KUKA KRL program: f1_Kuka_APT205T02S05.SRC

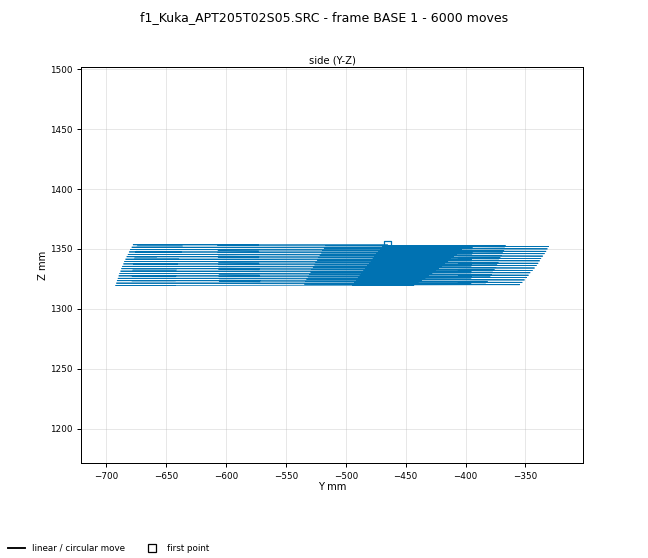
[picture p0: tool path of f1_Kuka_APT205T02S05.SRC in frame BASE 1, 6000 of 6001 moves have a stored position in this frame; points joined in program order, loops and branches not executed]
&ACCESS RVP
&REL 2
&PARAM TEMPLATE = C:\KRC\Roboter\Template\vorgabe
&PARAM EDITMASK = *
DEF f1_Kuka_APT205T02S05()


;FOLD INI;%{PE}%V3.2.0,%MKUKATPBASIS,%CINIT,%VCOMMON,%P
  ;FOLD BAS INI;%{E}%V3.2.0,%MKUKATPBASIS,%CINIT,%VINIT,%P
    GLOBAL INTERRUPT DECL 3 WHEN $STOPMESS==TRUE DO IR_STOPM ( )
    INTERRUPT ON 3
    BAS (#INITMOV,0 )
  ;ENDFOLD (BAS INI)
  ;FOLD USER INI;%{E}%V3.2.0,%MKUKATPUSER,%CINIT,%VINIT,%P
    ;Make your modifications here
  ;ENDFOLD (USER INI)
;ENDFOLD (INI)


;*** Make Null PTP Move
  PTP $pos_act

;*** Auto Load The Correct TOOL Data
  $tool=tool_data[2]

;*** Auto Load The Correct BASE Data
  $base=base_data[1]

  $ADVANCE = 5

;*** Restate Last Velocity
MMPM(30000.0)
SetRPM(8000)
LIN {X 0.183,Y -465.131,Z 1353.680,A 0.000,B 0.000,C 90.000,E1 158.284} C_DIS
LIN {X 0.167,Y -471.165,Z 1353.677,A 0.000,B 0.000,C 90.000,E1 157.794} C_DIS
LIN {X 0.121,Y -479.933,Z 1353.673,A 0.000,B 0.000,C 90.000,E1 157.050} C_DIS
LIN {X -0.013,Y -487.034,Z 1353.669,A 0.000,B 0.000,C 90.000,E1 156.433} C_DIS
LIN {X -0.242,Y -494.071,Z 1353.665,A 0.000,B 0.000,C 90.000,E1 155.793} C_DIS
LIN {X 0.180,Y -502.264,Z 1353.661,A 0.000,B 0.000,C 90.000,E1 154.921} C_DIS
LIN {X -0.273,Y -507.490,Z 1353.658,A 0.000,B 0.000,C 90.000,E1 154.409} C_DIS
LIN {X 0.116,Y -513.891,Z 1353.654,A 0.000,B 0.000,C 90.000,E1 153.640} C_DIS
LIN {X -0.118,Y -518.707,Z 1353.650,A 0.000,B 0.000,C 90.000,E1 153.076} C_DIS
LIN {X 0.081,Y -522.053,Z 1353.648,A 0.000,B 0.000,C 90.000,E1 152.615} C_DIS
LIN {X 0.144,Y -526.085,Z 1353.645,A 0.000,B 0.000,C 90.000,E1 152.025} C_DIS
LIN {X 0.240,Y -529.707,Z 1353.641,A 0.000,B 0.000,C 90.000,E1 151.435} C_DIS
LIN {X 0.217,Y -533.478,Z 1353.637,A 0.000,B 0.000,C 90.000,E1 150.717} C_DIS
LIN {X -0.096,Y -536.078,Z 1353.634,A 0.000,B 0.000,C 90.000,E1 150.177} C_DIS
LIN {X -0.207,Y -539.262,Z 1353.630,A 0.000,B 0.000,C 90.000,E1 149.331} C_DIS
LIN {X -0.021,Y -541.185,Z 1353.626,A 0.000,B 0.000,C 90.000,E1 148.742} C_DIS
LIN {X -0.285,Y -542.841,Z 1353.623,A 0.000,B 0.000,C 90.000,E1 148.201} C_DIS
LIN {X -0.054,Y -544.956,Z 1353.619,A 0.000,B 0.000,C 90.000,E1 147.327} C_DIS
LIN {X -0.260,Y -546.709,Z 1353.614,A 0.000,B 0.000,C 90.000,E1 146.501} C_DIS
LIN {X 0.272,Y -547.758,Z 1353.611,A 0.000,B 0.000,C 90.000,E1 145.881} C_DIS
LIN {X 0.097,Y -549.026,Z 1353.606,A 0.000,B 0.000,C 90.000,E1 145.055} C_DIS
LIN {X 0.251,Y -550.065,Z 1353.601,A 0.000,B 0.000,C 90.000,E1 144.196} C_DIS
LIN {X -0.292,Y -551.238,Z 1353.595,A 0.000,B 0.000,C 90.000,E1 143.130} C_DIS
LIN {X -0.048,Y -552.087,Z 1353.589,A 0.000,B 0.000,C 90.000,E1 141.984} C_DIS
LIN {X -0.168,Y -553.059,Z 1353.581,A 0.000,B 0.000,C 90.000,E1 140.598} C_DIS
LIN {X -0.278,Y -554.077,Z 1353.572,A 0.000,B 0.000,C 90.000,E1 138.933} C_DIS
LIN {X -0.078,Y -554.702,Z 1353.566,A 0.000,B 0.000,C 90.000,E1 137.796} C_DIS
LIN {X 0.097,Y -555.358,Z 1353.559,A 0.000,B 0.000,C 90.000,E1 136.662} C_DIS
LIN {X -0.235,Y -556.623,Z 1353.545,A 0.000,B 0.000,C 90.000,E1 134.190} C_DIS
LIN {X -0.134,Y -557.642,Z 1353.541,A 0.000,B 0.000,C 90.000,E1 133.299} C_DIS
LIN {X -0.120,Y -557.742,Z 1353.540,A 0.000,B 0.000,C 90.000,E1 133.257} C_DIS
LIN {X 0.206,Y -557.794,Z 1353.540,A 0.000,B 0.000,C 90.000,E1 133.218} C_DIS
LIN {X 0.099,Y -558.727,Z 1353.540,A 0.000,B 0.000,C 90.000,E1 133.137} C_DIS
LIN {X -0.091,Y -560.305,Z 1353.538,A 0.000,B 0.000,C 90.000,E1 132.894} C_DIS
LIN {X -0.316,Y -560.480,Z 1353.538,A 0.000,B 0.000,C 90.000,E1 132.852} C_DIS
LIN {X 0.022,Y -560.547,Z 1353.538,A 0.000,B 0.000,C 90.000,E1 132.813} C_DIS
LIN {X -0.018,Y -565.337,Z 1353.537,A 0.000,B 0.000,C 90.000,E1 132.609} C_DIS
LIN {X -0.209,Y -572.122,Z 1353.536,A 0.000,B 0.000,C 90.000,E1 132.447} C_DIS
LIN {X 0.152,Y -578.607,Z 1353.535,A 0.000,B 0.000,C 90.000,E1 132.204} C_DIS
LIN {X 0.195,Y -583.987,Z 1353.533,A 0.000,B 0.000,C 90.000,E1 131.919} C_DIS
LIN {X -0.113,Y -589.724,Z 1353.531,A 0.000,B 0.000,C 90.000,E1 131.595} C_DIS
LIN {X -0.223,Y -594.067,Z 1353.529,A 0.000,B 0.000,C 90.000,E1 131.310} C_DIS
LIN {X -0.123,Y -599.587,Z 1353.527,A 0.000,B 0.000,C 90.000,E1 130.862} C_DIS
LIN {X 0.104,Y -604.626,Z 1353.525,A 0.000,B 0.000,C 90.000,E1 130.415} C_DIS
LIN {X -0.052,Y -609.589,Z 1353.522,A 0.000,B 0.000,C 90.000,E1 129.967} C_DIS
LIN {X -0.137,Y -614.548,Z 1353.519,A 0.000,B 0.000,C 90.000,E1 129.483} C_DIS
LIN {X 0.107,Y -619.394,Z 1353.516,A 0.000,B 0.000,C 90.000,E1 128.955} C_DIS
LIN {X 0.250,Y -625.158,Z 1353.513,A 0.000,B 0.000,C 90.000,E1 128.302} C_DIS
LIN {X -0.237,Y -630.534,Z 1353.510,A 0.000,B 0.000,C 90.000,E1 127.729} C_DIS
LIN {X -0.014,Y -634.609,Z 1353.507,A 0.000,B 0.000,C 90.000,E1 127.202} C_DIS
LIN {X -0.289,Y -641.308,Z 1353.502,A 0.000,B 0.000,C 90.000,E1 126.377} C_DIS
LIN {X -0.064,Y -648.746,Z 1353.496,A 0.000,B 0.000,C 90.000,E1 125.358} C_DIS
LIN {X -0.070,Y -652.974,Z 1353.493,A 0.000,B 0.000,C 90.000,E1 124.739} C_DIS
LIN {X 0.045,Y -655.457,Z 1353.491,A 0.000,B 0.000,C 90.000,E1 124.358} C_DIS
LIN {X -0.290,Y -659.110,Z 1353.488,A 0.000,B 0.000,C 90.000,E1 123.785} C_DIS
LIN {X -0.210,Y -662.478,Z 1353.484,A 0.000,B 0.000,C 90.000,E1 123.166} C_DIS
LIN {X -0.165,Y -664.889,Z 1353.481,A 0.000,B 0.000,C 90.000,E1 122.673} C_DIS
LIN {X 0.027,Y -668.041,Z 1353.477,A 0.000,B 0.000,C 90.000,E1 121.926} C_DIS
LIN {X -0.101,Y -670.798,Z 1353.473,A 0.000,B 0.000,C 90.000,E1 121.209} C_DIS
LIN {X -0.265,Y -673.818,Z 1353.468,A 0.000,B 0.000,C 90.000,E1 120.256} C_DIS
LIN {X -0.330,Y -675.665,Z 1353.464,A 0.000,B 0.000,C 90.000,E1 119.539} C_DIS
LIN {X -0.374,Y -676.912,Z 1353.460,A 0.000,B 0.000,C 90.000,E1 118.821} C_DIS
LIN {X -0.404,Y -677.509,Z 1353.456,A 0.000,B 0.000,C 90.000,E1 118.103} C_DIS
LIN {X 0.173,Y -677.641,Z 1353.452,A 0.000,B 0.000,C 90.000,E1 117.334} C_DIS
LIN {X 0.338,Y -677.452,Z 1353.447,A 0.000,B 0.000,C 90.000,E1 116.360} C_DIS
LIN {X 0.010,Y -677.039,Z 1353.443,A 0.000,B 0.000,C 90.000,E1 115.668} C_DIS
LIN {X -0.034,Y -676.246,Z 1353.439,A 0.000,B 0.000,C 90.000,E1 114.951} C_DIS
LIN {X 0.055,Y -675.448,Z 1353.436,A 0.000,B 0.000,C 90.000,E1 114.463} C_DIS
LIN {X -0.195,Y -673.854,Z 1353.433,A 0.000,B 0.000,C 90.000,E1 114.003} C_DIS
LIN {X -0.289,Y -672.736,Z 1353.432,A 0.000,B 0.000,C 90.000,E1 113.770} C_DIS
LIN {X 0.053,Y -669.200,Z 1353.429,A 0.000,B 0.000,C 90.000,E1 113.259} C_DIS
LIN {X 0.132,Y -667.975,Z 1353.429,A 0.000,B 0.000,C 90.000,E1 113.131} C_DIS
LIN {X 0.067,Y -661.845,Z 1353.426,A 0.000,B 0.000,C 90.000,E1 112.717} C_DIS
LIN {X -0.202,Y -659.937,Z 1353.426,A 0.000,B 0.000,C 90.000,E1 112.642} C_DIS
LIN {X 0.198,Y -653.354,Z 1353.425,A 0.000,B 0.000,C 90.000,E1 112.386} C_DIS
LIN {X 0.212,Y -645.926,Z 1353.423,A 0.000,B 0.000,C 90.000,E1 112.206} C_DIS
LIN {X 0.189,Y -635.486,Z 1353.422,A 0.000,B 0.000,C 90.000,E1 111.972} C_DIS
LIN {X 0.137,Y -635.322,Z 1353.422,A 0.000,B 0.000,C 90.000,E1 111.972} C_DIS
LIN {X -0.263,Y -636.382,Z 1353.421,A 0.000,B 0.000,C 90.000,E1 111.844} C_DIS
LIN {X 0.284,Y -644.889,Z 1353.416,A 0.000,B 0.000,C 90.000,E1 110.791} C_DIS
LIN {X 0.217,Y -649.631,Z 1353.412,A 0.000,B 0.000,C 90.000,E1 110.174} C_DIS
LIN {X 0.007,Y -654.094,Z 1353.408,A 0.000,B 0.000,C 90.000,E1 109.450} C_DIS
LIN {X -0.159,Y -657.809,Z 1353.404,A 0.000,B 0.000,C 90.000,E1 108.725} C_DIS
LIN {X -0.293,Y -661.030,Z 1353.400,A 0.000,B 0.000,C 90.000,E1 108.000} C_DIS
LIN {X 0.141,Y -664.980,Z 1353.395,A 0.000,B 0.000,C 90.000,E1 106.985} C_DIS
LIN {X 0.157,Y -666.754,Z 1353.392,A 0.000,B 0.000,C 90.000,E1 106.496} C_DIS
LIN {X -0.083,Y -669.107,Z 1353.388,A 0.000,B 0.000,C 90.000,E1 105.788} C_DIS
LIN {X -0.158,Y -669.814,Z 1353.386,A 0.000,B 0.000,C 90.000,E1 105.552} C_DIS
LIN {X -0.190,Y -671.501,Z 1353.382,A 0.000,B 0.000,C 90.000,E1 104.828} C_DIS
LIN {X 0.331,Y -672.524,Z 1353.380,A 0.000,B 0.000,C 90.000,E1 104.300} C_DIS
LIN {X 0.209,Y -673.257,Z 1353.377,A 0.000,B 0.000,C 90.000,E1 103.828} C_DIS
LIN {X 0.035,Y -673.939,Z 1353.373,A 0.000,B 0.000,C 90.000,E1 103.119} C_DIS
LIN {X -0.081,Y -674.212,Z 1353.370,A 0.000,B 0.000,C 90.000,E1 102.647} C_DIS
LIN {X 0.267,Y -674.154,Z 1353.366,A 0.000,B 0.000,C 90.000,E1 101.895} C_DIS
LIN {X 0.096,Y -673.684,Z 1353.362,A 0.000,B 0.000,C 90.000,E1 101.186} C_DIS
LIN {X -0.026,Y -673.153,Z 1353.360,A 0.000,B 0.000,C 90.000,E1 100.715} C_DIS
LIN {X -0.211,Y -672.846,Z 1353.358,A 0.000,B 0.000,C 90.000,E1 100.489} C_DIS
LIN {X 0.321,Y -671.939,Z 1353.356,A 0.000,B 0.000,C 90.000,E1 99.962} C_DIS
LIN {X 0.069,Y -670.767,Z 1353.353,A 0.000,B 0.000,C 90.000,E1 99.500} C_DIS
LIN {X -0.003,Y -670.111,Z 1353.352,A 0.000,B 0.000,C 90.000,E1 99.265} C_DIS
LIN {X -0.261,Y -668.546,Z 1353.349,A 0.000,B 0.000,C 90.000,E1 98.803} C_DIS
LIN {X 0.230,Y -666.752,Z 1353.346,A 0.000,B 0.000,C 90.000,E1 98.276} C_DIS
LIN {X -0.236,Y -663.690,Z 1353.342,A 0.000,B 0.000,C 90.000,E1 97.587} C_DIS
LIN {X 0.114,Y -660.735,Z 1353.339,A 0.000,B 0.000,C 90.000,E1 96.947} C_DIS
LIN {X 0.151,Y -656.334,Z 1353.334,A 0.000,B 0.000,C 90.000,E1 96.087} C_DIS
LIN {X -0.295,Y -652.814,Z 1353.331,A 0.000,B 0.000,C 90.000,E1 95.511} C_DIS
LIN {X -0.282,Y -647.351,Z 1353.326,A 0.000,B 0.000,C 90.000,E1 94.645} C_DIS
LIN {X -0.274,Y -642.136,Z 1353.322,A 0.000,B 0.000,C 90.000,E1 93.898} C_DIS
LIN {X -0.111,Y -638.342,Z 1353.319,A 0.000,B 0.000,C 90.000,E1 93.383} C_DIS
LIN {X -0.031,Y -632.660,Z 1353.315,A 0.000,B 0.000,C 90.000,E1 92.751} C_DIS
LIN {X -0.038,Y -622.818,Z 1353.310,A 0.000,B 0.000,C 90.000,E1 91.776} C_DIS
LIN {X 0.147,Y -616.480,Z 1353.307,A 0.000,B 0.000,C 90.000,E1 91.146} C_DIS
LIN {X -0.106,Y -609.537,Z 1353.303,A 0.000,B 0.000,C 90.000,E1 90.573} C_DIS
LIN {X 0.254,Y -603.296,Z 1353.301,A 0.000,B 0.000,C 90.000,E1 90.115} C_DIS
LIN {X 0.236,Y -598.176,Z 1353.299,A 0.000,B 0.000,C 90.000,E1 89.828} C_DIS
LIN {X 0.187,Y -594.693,Z 1353.298,A 0.000,B 0.000,C 90.000,E1 89.656} C_DIS
LIN {X 0.205,Y -581.240,Z 1353.295,A 0.000,B 0.000,C 90.000,E1 89.083} C_DIS
LIN {X 0.020,Y -578.376,Z 1353.294,A 0.000,B 0.000,C 90.000,E1 88.969} C_DIS
LIN {X 0.191,Y -575.836,Z 1353.293,A 0.000,B 0.000,C 90.000,E1 88.797} C_DIS
LIN {X -0.266,Y -574.481,Z 1353.293,A 0.000,B 0.000,C 90.000,E1 88.740} C_DIS
LIN {X -0.147,Y -573.606,Z 1353.292,A 0.000,B 0.000,C 90.000,E1 88.625} C_DIS
LIN {X -0.152,Y -573.255,Z 1353.292,A 0.000,B 0.000,C 90.000,E1 88.568} C_DIS
LIN {X -0.137,Y -573.024,Z 1353.291,A 0.000,B 0.000,C 90.000,E1 88.453} C_DIS
LIN {X -0.080,Y -572.878,Z 1353.290,A 0.000,B 0.000,C 90.000,E1 88.165} C_DIS
LIN {X -0.016,Y -573.318,Z 1353.286,A 0.000,B 0.000,C 90.000,E1 87.478} C_DIS
LIN {X -0.115,Y -575.111,Z 1353.275,A 0.000,B 0.000,C 90.000,E1 85.584} C_DIS
LIN {X 0.078,Y -577.539,Z 1353.263,A 0.000,B 0.000,C 90.000,E1 83.394} C_DIS
LIN {X -0.026,Y -579.410,Z 1353.254,A 0.000,B 0.000,C 90.000,E1 81.781} C_DIS
LIN {X -0.153,Y -581.083,Z 1353.247,A 0.000,B 0.000,C 90.000,E1 80.443} C_DIS
LIN {X 0.090,Y -582.298,Z 1353.241,A 0.000,B 0.000,C 90.000,E1 79.342} C_DIS
LIN {X 0.124,Y -583.632,Z 1353.233,A 0.000,B 0.000,C 90.000,E1 77.993} C_DIS
LIN {X 0.184,Y -584.854,Z 1353.226,A 0.000,B 0.000,C 90.000,E1 76.645} C_DIS
LIN {X -0.165,Y -585.974,Z 1353.219,A 0.000,B 0.000,C 90.000,E1 75.338} C_DIS
LIN {X -0.169,Y -586.736,Z 1353.213,A 0.000,B 0.000,C 90.000,E1 74.267} C_DIS
LIN {X 0.165,Y -587.915,Z 1353.202,A 0.000,B 0.000,C 90.000,E1 72.362} C_DIS
LIN {X 0.031,Y -588.687,Z 1353.195,A 0.000,B 0.000,C 90.000,E1 71.040} C_DIS
LIN {X -0.023,Y -589.671,Z 1353.186,A 0.000,B 0.000,C 90.000,E1 69.444} C_DIS
LIN {X -0.059,Y -591.222,Z 1353.172,A 0.000,B 0.000,C 90.000,E1 67.050} C_DIS
LIN {X 0.057,Y -592.676,Z 1353.162,A 0.000,B 0.000,C 90.000,E1 65.177} C_DIS
LIN {X -0.334,Y -593.414,Z 1353.156,A 0.000,B 0.000,C 90.000,E1 64.152} C_DIS
LIN {X -0.004,Y -594.376,Z 1353.149,A 0.000,B 0.000,C 90.000,E1 62.794} C_DIS
LIN {X 0.081,Y -596.127,Z 1353.137,A 0.000,B 0.000,C 90.000,E1 60.667} C_DIS
LIN {X 0.272,Y -598.255,Z 1353.125,A 0.000,B 0.000,C 90.000,E1 58.535} C_DIS
LIN {X 0.185,Y -599.776,Z 1353.117,A 0.000,B 0.000,C 90.000,E1 56.962} C_DIS
LIN {X -0.018,Y -600.796,Z 1353.111,A 0.000,B 0.000,C 90.000,E1 55.928} C_DIS
LIN {X 0.038,Y -602.054,Z 1353.103,A 0.000,B 0.000,C 90.000,E1 54.609} C_DIS
LIN {X 0.136,Y -603.753,Z 1353.093,A 0.000,B 0.000,C 90.000,E1 52.763} C_DIS
LIN {X -0.152,Y -604.595,Z 1353.087,A 0.000,B 0.000,C 90.000,E1 51.743} C_DIS
LIN {X 0.092,Y -605.607,Z 1353.079,A 0.000,B 0.000,C 90.000,E1 50.150} C_DIS
LIN {X 0.207,Y -606.155,Z 1353.073,A 0.000,B 0.000,C 90.000,E1 49.094} C_DIS
LIN {X -0.124,Y -606.527,Z 1353.067,A 0.000,B 0.000,C 90.000,E1 48.081} C_DIS
LIN {X -0.192,Y -606.838,Z 1353.060,A 0.000,B 0.000,C 90.000,E1 46.782} C_DIS
LIN {X -0.042,Y -606.960,Z 1353.051,A 0.000,B 0.000,C 90.000,E1 45.202} C_DIS
LIN {X -0.368,Y -606.826,Z 1353.045,A 0.000,B 0.000,C 90.000,E1 44.190} C_DIS
LIN {X 0.171,Y -606.456,Z 1353.040,A 0.000,B 0.000,C 90.000,E1 43.095} C_DIS
LIN {X -0.087,Y -605.775,Z 1353.031,A 0.000,B 0.000,C 90.000,E1 41.553} C_DIS
LIN {X 0.038,Y -605.198,Z 1353.025,A 0.000,B 0.000,C 90.000,E1 40.496} C_DIS
LIN {X 0.206,Y -604.342,Z 1353.016,A 0.000,B 0.000,C 90.000,E1 38.910} C_DIS
LIN {X 0.181,Y -603.425,Z 1353.009,A 0.000,B 0.000,C 90.000,E1 37.604} C_DIS
LIN {X -0.115,Y -602.354,Z 1353.003,A 0.000,B 0.000,C 90.000,E1 36.583} C_DIS
LIN {X 0.391,Y -601.707,Z 1353.000,A 0.000,B 0.000,C 90.000,E1 36.011} C_DIS
LIN {X 0.299,Y -600.464,Z 1352.996,A 0.000,B 0.000,C 90.000,E1 35.231} C_DIS
LIN {X 0.093,Y -598.433,Z 1352.990,A 0.000,B 0.000,C 90.000,E1 34.199} C_DIS
LIN {X -0.037,Y -596.783,Z 1352.986,A 0.000,B 0.000,C 90.000,E1 33.420} C_DIS
LIN {X 0.205,Y -594.246,Z 1352.980,A 0.000,B 0.000,C 90.000,E1 32.339} C_DIS
LIN {X 0.210,Y -592.058,Z 1352.975,A 0.000,B 0.000,C 90.000,E1 31.544} C_DIS
LIN {X -0.122,Y -588.527,Z 1352.969,A 0.000,B 0.000,C 90.000,E1 30.512} C_DIS
LIN {X 0.158,Y -586.676,Z 1352.967,A 0.000,B 0.000,C 90.000,E1 29.951} C_DIS
LIN {X 0.090,Y -583.481,Z 1352.962,A 0.000,B 0.000,C 90.000,E1 29.155} C_DIS
LIN {X -0.151,Y -578.574,Z 1352.956,A 0.000,B 0.000,C 90.000,E1 28.103} C_DIS
LIN {X 0.037,Y -573.018,Z 1352.950,A 0.000,B 0.000,C 90.000,E1 27.001} C_DIS
LIN {X 0.145,Y -569.164,Z 1352.946,A 0.000,B 0.000,C 90.000,E1 26.309} C_DIS
LIN {X 0.047,Y -565.823,Z 1352.943,A 0.000,B 0.000,C 90.000,E1 25.771} C_DIS
LIN {X 0.091,Y -561.388,Z 1352.939,A 0.000,B 0.000,C 90.000,E1 25.079} C_DIS
LIN {X 0.300,Y -558.527,Z 1352.937,A 0.000,B 0.000,C 90.000,E1 24.643} C_DIS
LIN {X 0.279,Y -553.466,Z 1352.933,A 0.000,B 0.000,C 90.000,E1 23.951} C_DIS
LIN {X 0.211,Y -548.153,Z 1352.929,A 0.000,B 0.000,C 90.000,E1 23.259} C_DIS
LIN {X -0.105,Y -542.387,Z 1352.926,A 0.000,B 0.000,C 90.000,E1 22.589} C_DIS
LIN {X -0.051,Y -533.794,Z 1352.920,A 0.000,B 0.000,C 90.000,E1 21.589} C_DIS
LIN {X -0.220,Y -523.413,Z 1352.914,A 0.000,B 0.000,C 90.000,E1 20.482} C_DIS
LIN {X 0.087,Y -511.582,Z 1352.907,A 0.000,B 0.000,C 90.000,E1 19.214} C_DIS
LIN {X -0.134,Y -503.938,Z 1352.902,A 0.000,B 0.000,C 90.000,E1 18.417} C_DIS
LIN {X 0.088,Y -493.051,Z 1352.896,A 0.000,B 0.000,C 90.000,E1 17.275} C_DIS
LIN {X 0.155,Y -482.910,Z 1352.891,A 0.000,B 0.000,C 90.000,E1 16.315} C_DIS
LIN {X -0.050,Y -466.107,Z 1352.882,A 0.000,B 0.000,C 90.000,E1 14.717} C_DIS
LIN {X -0.017,Y -454.626,Z 1352.875,A 0.000,B 0.000,C 90.000,E1 13.592} C_DIS
LIN {X 0.099,Y -434.707,Z 1352.864,A 0.000,B 0.000,C 90.000,E1 11.535} C_DIS
LIN {X 0.038,Y -419.253,Z 1352.855,A 0.000,B 0.000,C 90.000,E1 9.849} C_DIS
LIN {X 0.108,Y -408.120,Z 1352.848,A 0.000,B 0.000,C 90.000,E1 8.568} C_DIS
LIN {X 0.156,Y -399.605,Z 1352.842,A 0.000,B 0.000,C 90.000,E1 7.587} C_DIS
LIN {X -0.151,Y -396.843,Z 1352.840,A 0.000,B 0.000,C 90.000,E1 7.296} C_DIS
LIN {X -0.035,Y -394.063,Z 1352.838,A 0.000,B 0.000,C 90.000,E1 6.834} C_DIS
LIN {X -0.072,Y -394.049,Z 1352.838,A 0.000,B 0.000,C 90.000,E1 6.834} C_DIS
LIN {X 0.040,Y -394.965,Z 1352.837,A 0.000,B 0.000,C 90.000,E1 6.663} C_DIS
LIN {X -0.100,Y -398.981,Z 1352.835,A 0.000,B 0.000,C 90.000,E1 6.315} C_DIS
LIN {X -0.090,Y -412.650,Z 1352.830,A 0.000,B 0.000,C 90.000,E1 5.334} C_DIS
LIN {X -0.158,Y -415.923,Z 1352.828,A 0.000,B 0.000,C 90.000,E1 5.106} C_DIS
LIN {X -0.168,Y -423.370,Z 1352.825,A 0.000,B 0.000,C 90.000,E1 4.473} C_DIS
LIN {X -0.125,Y -429.177,Z 1352.822,A 0.000,B 0.000,C 90.000,E1 3.898} C_DIS
LIN {X -0.204,Y -436.191,Z 1352.817,A 0.000,B 0.000,C 90.000,E1 3.151} C_DIS
LIN {X -0.062,Y -442.966,Z 1352.813,A 0.000,B 0.000,C 90.000,E1 2.350} C_DIS
LIN {X -0.089,Y -448.332,Z 1352.810,A 0.000,B 0.000,C 90.000,E1 1.718} C_DIS
LIN {X -0.125,Y -454.577,Z 1352.805,A 0.000,B 0.000,C 90.000,E1 0.917} C_DIS
LIN {X -0.227,Y -459.308,Z 1352.802,A 0.000,B 0.000,C 90.000,E1 0.286} C_DIS
LIN {X 0.027,Y -465.795,Z 1352.796,A 0.000,B 0.000,C 90.000,E1 359.312} C_DIS
LIN {X 0.129,Y -470.852,Z 1352.792,A 0.000,B 0.000,C 90.000,E1 358.511} C_DIS
LIN {X -0.047,Y -476.329,Z 1352.787,A 0.000,B 0.000,C 90.000,E1 357.593} C_DIS
LIN {X 0.014,Y -479.818,Z 1352.783,A 0.000,B 0.000,C 90.000,E1 356.963} C_DIS
LIN {X -0.209,Y -483.851,Z 1352.779,A 0.000,B 0.000,C 90.000,E1 356.216} C_DIS
LIN {X -0.062,Y -486.825,Z 1352.776,A 0.000,B 0.000,C 90.000,E1 355.584} C_DIS
LIN {X -0.221,Y -490.207,Z 1352.771,A 0.000,B 0.000,C 90.000,E1 354.837} C_DIS
LIN {X -0.024,Y -492.765,Z 1352.768,A 0.000,B 0.000,C 90.000,E1 354.204} C_DIS
LIN {X 0.088,Y -496.185,Z 1352.763,A 0.000,B 0.000,C 90.000,E1 353.280} C_DIS
LIN {X 0.239,Y -499.354,Z 1352.758,A 0.000,B 0.000,C 90.000,E1 352.356} C_DIS
LIN {X 0.156,Y -500.373,Z 1352.756,A 0.000,B 0.000,C 90.000,E1 352.064} C_DIS
LIN {X -0.143,Y -502.907,Z 1352.751,A 0.000,B 0.000,C 90.000,E1 351.197} C_DIS
LIN {X 0.078,Y -505.288,Z 1352.746,A 0.000,B 0.000,C 90.000,E1 350.274} C_DIS
LIN {X -0.139,Y -508.072,Z 1352.739,A 0.000,B 0.000,C 90.000,E1 349.106} C_DIS
LIN {X 0.224,Y -509.966,Z 1352.734,A 0.000,B 0.000,C 90.000,E1 348.173} C_DIS
LIN {X 0.108,Y -511.644,Z 1352.729,A 0.000,B 0.000,C 90.000,E1 347.297} C_DIS
LIN {X 0.124,Y -513.042,Z 1352.725,A 0.000,B 0.000,C 90.000,E1 346.408} C_DIS
LIN {X 0.133,Y -514.692,Z 1352.718,A 0.000,B 0.000,C 90.000,E1 345.227} C_DIS
LIN {X 0.188,Y -515.655,Z 1352.713,A 0.000,B 0.000,C 90.000,E1 344.338} C_DIS
LIN {X -0.244,Y -516.324,Z 1352.708,A 0.000,B 0.000,C 90.000,E1 343.504} C_DIS
LIN {X -0.024,Y -516.755,Z 1352.703,A 0.000,B 0.000,C 90.000,E1 342.598} C_DIS
LIN {X 0.042,Y -516.921,Z 1352.698,A 0.000,B 0.000,C 90.000,E1 341.710} C_DIS
LIN {X -0.222,Y -516.779,Z 1352.694,A 0.000,B 0.000,C 90.000,E1 340.859} C_DIS
LIN {X -0.090,Y -516.613,Z 1352.692,A 0.000,B 0.000,C 90.000,E1 340.550} C_DIS
LIN {X 0.043,Y -516.273,Z 1352.690,A 0.000,B 0.000,C 90.000,E1 340.242} C_DIS
LIN {X 0.176,Y -515.763,Z 1352.689,A 0.000,B 0.000,C 90.000,E1 339.934} C_DIS
LIN {X 0.130,Y -514.975,Z 1352.687,A 0.000,B 0.000,C 90.000,E1 339.645} C_DIS
LIN {X -0.223,Y -513.741,Z 1352.685,A 0.000,B 0.000,C 90.000,E1 339.390} C_DIS
LIN {X 0.081,Y -512.783,Z 1352.685,A 0.000,B 0.000,C 90.000,E1 339.209} C_DIS
LIN {X -0.095,Y -510.810,Z 1352.684,A 0.000,B 0.000,C 90.000,E1 339.082} C_DIS
LIN {X -0.228,Y -481.772,Z 1352.677,A 0.000,B 0.000,C 90.000,E1 337.794} C_DIS
LIN {X 0.049,Y -453.227,Z 1352.668,A 0.000,B 0.000,C 90.000,E1 336.305} C_DIS
LIN {X 0.187,Y -428.324,Z 1352.660,A 0.000,B 0.000,C 90.000,E1 334.845} C_DIS
LIN {X -0.103,Y -405.367,Z 1352.652,A 0.000,B 0.000,C 90.000,E1 333.384} C_DIS
LIN {X 0.001,Y -384.338,Z 1352.643,A 0.000,B 0.000,C 90.000,E1 331.820} C_DIS
LIN {X 0.190,Y -366.662,Z 1352.635,A 0.000,B 0.000,C 90.000,E1 330.333} C_DIS
LIN {X 0.162,Y -366.645,Z 1352.635,A 0.000,B 0.000,C 90.000,E1 330.333} C_DIS
LIN {X -0.069,Y -371.456,Z 1352.603,A 0.000,B 0.000,C 90.000,E1 324.562} C_DIS
LIN {X -0.081,Y -371.815,Z 1352.601,A 0.000,B 0.000,C 90.000,E1 324.196} C_DIS
LIN {X -0.013,Y -377.467,Z 1352.567,A 0.000,B 0.000,C 90.000,E1 317.957} C_DIS
LIN {X -0.027,Y -377.945,Z 1352.564,A 0.000,B 0.000,C 90.000,E1 317.595} C_DIS
LIN {X 0.001,Y -378.528,Z 1352.560,A 0.000,B 0.000,C 90.000,E1 316.863} C_DIS
LIN {X 0.023,Y -384.552,Z 1352.528,A 0.000,B 0.000,C 90.000,E1 311.067} C_DIS
LIN {X 0.068,Y -384.947,Z 1352.526,A 0.000,B 0.000,C 90.000,E1 310.701} C_DIS
LIN {X 0.016,Y -390.724,Z 1352.494,A 0.000,B 0.000,C 90.000,E1 304.978} C_DIS
LIN {X 0.083,Y -391.221,Z 1352.492,A 0.000,B 0.000,C 90.000,E1 304.612} C_DIS
LIN {X -0.110,Y -396.934,Z 1352.459,A 0.000,B 0.000,C 90.000,E1 298.615} C_DIS
LIN {X 0.190,Y -401.301,Z 1352.428,A 0.000,B 0.000,C 90.000,E1 292.950} C_DIS
LIN {X -0.100,Y -401.646,Z 1352.426,A 0.000,B 0.000,C 90.000,E1 292.642} C_DIS
LIN {X 0.036,Y -404.726,Z 1352.395,A 0.000,B 0.000,C 90.000,E1 287.040} C_DIS
LIN {X 0.039,Y -406.144,Z 1352.364,A 0.000,B 0.000,C 90.000,E1 281.478} C_DIS
LIN {X 0.137,Y -405.687,Z 1352.333,A 0.000,B 0.000,C 90.000,E1 275.910} C_DIS
LIN {X -0.195,Y -403.571,Z 1352.306,A 0.000,B 0.000,C 90.000,E1 271.088} C_DIS
LIN {X 0.144,Y -403.221,Z 1352.302,A 0.000,B 0.000,C 90.000,E1 270.344} C_DIS
LIN {X -0.022,Y -399.083,Z 1352.273,A 0.000,B 0.000,C 90.000,E1 265.122} C_DIS
LIN {X -0.080,Y -398.829,Z 1352.271,A 0.000,B 0.000,C 90.000,E1 264.780} C_DIS
LIN {X 0.206,Y -393.321,Z 1352.244,A 0.000,B 0.000,C 90.000,E1 259.803} C_DIS
LIN {X 0.127,Y -392.730,Z 1352.240,A 0.000,B 0.000,C 90.000,E1 259.106} C_DIS
LIN {X -0.180,Y -386.288,Z 1352.214,A 0.000,B 0.000,C 90.000,E1 254.519} C_DIS
LIN {X -0.109,Y -385.187,Z 1352.208,A 0.000,B 0.000,C 90.000,E1 253.433} C_DIS
LIN {X -0.142,Y -382.701,Z 1352.200,A 0.000,B 0.000,C 90.000,E1 252.000} C_DIS
LIN {X 0.113,Y -376.547,Z 1352.176,A 0.000,B 0.000,C 90.000,E1 247.614} C_DIS
LIN {X -0.109,Y -376.137,Z 1352.174,A 0.000,B 0.000,C 90.000,E1 247.283} C_DIS
LIN {X 0.063,Y -368.301,Z 1352.147,A 0.000,B 0.000,C 90.000,E1 242.487} C_DIS
LIN {X 0.100,Y -366.444,Z 1352.139,A 0.000,B 0.000,C 90.000,E1 241.001} C_DIS
LIN {X -0.135,Y -365.880,Z 1352.137,A 0.000,B 0.000,C 90.000,E1 240.667} C_DIS
LIN {X -0.046,Y -359.073,Z 1352.114,A 0.000,B 0.000,C 90.000,E1 236.548} C_DIS
LIN {X 0.042,Y -356.223,Z 1352.102,A 0.000,B 0.000,C 90.000,E1 234.276} C_DIS
LIN {X -0.028,Y -355.681,Z 1352.099,A 0.000,B 0.000,C 90.000,E1 233.909} C_DIS
LIN {X 0.041,Y -348.681,Z 1352.074,A 0.000,B 0.000,C 90.000,E1 229.337} C_DIS
LIN {X -0.149,Y -346.095,Z 1352.061,A 0.000,B 0.000,C 90.000,E1 227.067} C_DIS
LIN {X -0.010,Y -339.726,Z 1352.036,A 0.000,B 0.000,C 90.000,E1 222.405} C_DIS
LIN {X 0.032,Y -336.726,Z 1352.018,A 0.000,B 0.000,C 90.000,E1 219.277} C_DIS
LIN {X 0.136,Y -330.657,Z 1351.987,A 0.000,B 0.000,C 90.000,E1 213.579} C_DIS
LIN {X 0.010,Y -330.641,Z 1351.987,A 0.000,B 0.000,C 90.000,E1 213.579} C_DIS
LIN {X -0.007,Y -330.667,Z 1351.987,A 0.000,B 0.000,C 90.000,E1 213.579} C_DIS
LIN {X -0.087,Y -348.232,Z 1351.976,A 0.000,B 0.000,C 90.000,E1 211.750} C_DIS
LIN {X -0.025,Y -367.506,Z 1351.966,A 0.000,B 0.000,C 90.000,E1 209.951} C_DIS
LIN {X -0.168,Y -387.102,Z 1351.958,A 0.000,B 0.000,C 90.000,E1 208.359} C_DIS
LIN {X 0.106,Y -408.632,Z 1351.949,A 0.000,B 0.000,C 90.000,E1 206.744} C_DIS
LIN {X 0.218,Y -432.130,Z 1351.940,A 0.000,B 0.000,C 90.000,E1 205.207} C_DIS
LIN {X 0.040,Y -447.345,Z 1351.935,A 0.000,B 0.000,C 90.000,E1 204.335} C_DIS
LIN {X 0.103,Y -449.075,Z 1351.934,A 0.000,B 0.000,C 90.000,E1 204.131} C_DIS
LIN {X -0.119,Y -449.941,Z 1351.933,A 0.000,B 0.000,C 90.000,E1 204.003} C_DIS
LIN {X 0.071,Y -450.638,Z 1351.932,A 0.000,B 0.000,C 90.000,E1 203.823} C_DIS
LIN {X -0.050,Y -451.762,Z 1351.931,A 0.000,B 0.000,C 90.000,E1 203.515} C_DIS
LIN {X -0.167,Y -452.616,Z 1351.929,A 0.000,B 0.000,C 90.000,E1 203.206} C_DIS
LIN {X -0.280,Y -453.319,Z 1351.927,A 0.000,B 0.000,C 90.000,E1 202.898} C_DIS
LIN {X 0.097,Y -454.325,Z 1351.923,A 0.000,B 0.000,C 90.000,E1 202.206} C_DIS
LIN {X 0.113,Y -455.783,Z 1351.916,A 0.000,B 0.000,C 90.000,E1 200.918} C_DIS
LIN {X 0.152,Y -457.089,Z 1351.909,A 0.000,B 0.000,C 90.000,E1 199.631} C_DIS
LIN {X -0.271,Y -459.133,Z 1351.899,A 0.000,B 0.000,C 90.000,E1 197.764} C_DIS
LIN {X 0.010,Y -460.583,Z 1351.890,A 0.000,B 0.000,C 90.000,E1 196.134} C_DIS
LIN {X 0.272,Y -461.683,Z 1351.883,A 0.000,B 0.000,C 90.000,E1 194.828} C_DIS
LIN {X -0.069,Y -463.574,Z 1351.870,A 0.000,B 0.000,C 90.000,E1 192.647} C_DIS
LIN {X -0.014,Y -465.592,Z 1351.858,A 0.000,B 0.000,C 90.000,E1 190.423} C_DIS
LIN {X -0.148,Y -466.802,Z 1351.849,A 0.000,B 0.000,C 90.000,E1 188.859} C_DIS
LIN {X -0.061,Y -467.701,Z 1351.842,A 0.000,B 0.000,C 90.000,E1 187.587} C_DIS
LIN {X -0.159,Y -468.471,Z 1351.833,A 0.000,B 0.000,C 90.000,E1 186.024} C_DIS
LIN {X 0.123,Y -468.966,Z 1351.825,A 0.000,B 0.000,C 90.000,E1 184.416} C_DIS
LIN {X -0.080,Y -469.217,Z 1351.819,A 0.000,B 0.000,C 90.000,E1 183.498} C_DIS
LIN {X -0.042,Y -469.187,Z 1351.813,A 0.000,B 0.000,C 90.000,E1 182.236} C_DIS
LIN {X 0.222,Y -469.011,Z 1351.807,A 0.000,B 0.000,C 90.000,E1 181.260} C_DIS
LIN {X 0.002,Y -468.506,Z 1351.802,A 0.000,B 0.000,C 90.000,E1 180.344} C_DIS
LIN {X 0.010,Y -468.041,Z 1351.798,A 0.000,B 0.000,C 90.000,E1 179.714} C_DIS
LIN {X 0.011,Y -466.576,Z 1351.792,A 0.000,B 0.000,C 90.000,E1 178.453} C_DIS
LIN {X -0.222,Y -465.386,Z 1351.786,A 0.000,B 0.000,C 90.000,E1 177.535} C_DIS
LIN {X 0.001,Y -463.836,Z 1351.781,A 0.000,B 0.000,C 90.000,E1 176.560} C_DIS
LIN {X -0.004,Y -462.565,Z 1351.777,A 0.000,B 0.000,C 90.000,E1 175.927} C_DIS
LIN {X 0.182,Y -460.315,Z 1351.772,A 0.000,B 0.000,C 90.000,E1 174.951} C_DIS
LIN {X 0.151,Y -458.478,Z 1351.769,A 0.000,B 0.000,C 90.000,E1 174.318} C_DIS
LIN {X 0.016,Y -456.792,Z 1351.766,A 0.000,B 0.000,C 90.000,E1 173.856} C_DIS
LIN {X -0.045,Y -454.202,Z 1351.762,A 0.000,B 0.000,C 90.000,E1 173.223} C_DIS
LIN {X -0.128,Y -451.329,Z 1351.759,A 0.000,B 0.000,C 90.000,E1 172.591} C_DIS
LIN {X 0.016,Y -446.330,Z 1351.753,A 0.000,B 0.000,C 90.000,E1 171.602} C_DIS
LIN {X 0.032,Y -440.311,Z 1351.748,A 0.000,B 0.000,C 90.000,E1 170.622} C_DIS
LIN {X -0.151,Y -430.178,Z 1351.740,A 0.000,B 0.000,C 90.000,E1 169.162} C_DIS
LIN {X -0.168,Y -422.153,Z 1351.733,A 0.000,B 0.000,C 90.000,E1 167.993} C_DIS
LIN {X -0.153,Y -412.271,Z 1351.725,A 0.000,B 0.000,C 90.000,E1 166.464} C_DIS
LIN {X 0.020,Y -405.870,Z 1351.719,A 0.000,B 0.000,C 90.000,E1 165.408} C_DIS
LIN {X 0.120,Y -402.746,Z 1351.715,A 0.000,B 0.000,C 90.000,E1 164.700} C_DIS
LIN {X 0.167,Y -402.223,Z 1351.714,A 0.000,B 0.000,C 90.000,E1 164.519} C_DIS
LIN {X -0.148,Y -401.357,Z 1351.710,A 0.000,B 0.000,C 90.000,E1 163.866} C_DIS
LIN {X -0.183,Y -401.776,Z 1351.710,A 0.000,B 0.000,C 90.000,E1 163.740} C_DIS
LIN {X -0.015,Y -404.556,Z 1351.707,A 0.000,B 0.000,C 90.000,E1 163.323} C_DIS
LIN {X 0.083,Y -407.541,Z 1351.705,A 0.000,B 0.000,C 90.000,E1 162.960} C_DIS
LIN {X -0.146,Y -411.501,Z 1351.703,A 0.000,B 0.000,C 90.000,E1 162.598} C_DIS
LIN {X 0.067,Y -417.594,Z 1351.700,A 0.000,B 0.000,C 90.000,E1 162.000} C_DIS
LIN {X 0.052,Y -423.966,Z 1351.697,A 0.000,B 0.000,C 90.000,E1 161.456} C_DIS
LIN {X -0.171,Y -444.601,Z 1351.688,A 0.000,B 0.000,C 90.000,E1 159.880} C_DIS
LIN {X -0.018,Y -457.288,Z 1351.683,A 0.000,B 0.000,C 90.000,E1 158.901} C_DIS
LIN {X 0.131,Y -466.519,Z 1351.679,A 0.000,B 0.000,C 90.000,E1 158.156} C_DIS
LIN {X 0.062,Y -471.041,Z 1351.677,A 0.000,B 0.000,C 90.000,E1 157.794} C_DIS
LIN {X 0.074,Y -479.801,Z 1351.673,A 0.000,B 0.000,C 90.000,E1 157.050} C_DIS
LIN {X 0.030,Y -487.055,Z 1351.669,A 0.000,B 0.000,C 90.000,E1 156.410} C_DIS
LIN {X 0.097,Y -494.071,Z 1351.665,A 0.000,B 0.000,C 90.000,E1 155.741} C_DIS
LIN {X 0.148,Y -500.907,Z 1351.661,A 0.000,B 0.000,C 90.000,E1 155.049} C_DIS
LIN {X -0.159,Y -504.908,Z 1351.659,A 0.000,B 0.000,C 90.000,E1 154.665} C_DIS
LIN {X -0.052,Y -509.945,Z 1351.656,A 0.000,B 0.000,C 90.000,E1 154.101} C_DIS
LIN {X -0.001,Y -514.978,Z 1351.653,A 0.000,B 0.000,C 90.000,E1 153.512} C_DIS
LIN {X -0.060,Y -518.580,Z 1351.650,A 0.000,B 0.000,C 90.000,E1 153.076} C_DIS
LIN {X 0.138,Y -521.928,Z 1351.648,A 0.000,B 0.000,C 90.000,E1 152.615} C_DIS
LIN {X 0.201,Y -525.967,Z 1351.645,A 0.000,B 0.000,C 90.000,E1 152.025} C_DIS
LIN {X 0.043,Y -529.594,Z 1351.641,A 0.000,B 0.000,C 90.000,E1 151.463} C_DIS
LIN {X 0.273,Y -533.381,Z 1351.638,A 0.000,B 0.000,C 90.000,E1 150.717} C_DIS
LIN {X -0.308,Y -535.916,Z 1351.634,A 0.000,B 0.000,C 90.000,E1 150.205} C_DIS
LIN {X -0.154,Y -539.110,Z 1351.630,A 0.000,B 0.000,C 90.000,E1 149.331} C_DIS
LIN {X 0.031,Y -540.980,Z 1351.626,A 0.000,B 0.000,C 90.000,E1 148.742} C_DIS
LIN {X -0.234,Y -542.665,Z 1351.623,A 0.000,B 0.000,C 90.000,E1 148.201} C_DIS
LIN {X -0.005,Y -544.766,Z 1351.619,A 0.000,B 0.000,C 90.000,E1 147.327} C_DIS
LIN {X -0.212,Y -546.523,Z 1351.614,A 0.000,B 0.000,C 90.000,E1 146.501} C_DIS
LIN {X -0.091,Y -547.989,Z 1351.609,A 0.000,B 0.000,C 90.000,E1 145.642} C_DIS
LIN {X 0.189,Y -549.199,Z 1351.604,A 0.000,B 0.000,C 90.000,E1 144.769} C_DIS
LIN {X 0.077,Y -550.477,Z 1351.598,A 0.000,B 0.000,C 90.000,E1 143.657} C_DIS
LIN {X -0.194,Y -551.266,Z 1351.594,A 0.000,B 0.000,C 90.000,E1 142.844} C_DIS
LIN {X -0.012,Y -551.894,Z 1351.589,A 0.000,B 0.000,C 90.000,E1 141.984} C_DIS
LIN {X -0.135,Y -552.830,Z 1351.581,A 0.000,B 0.000,C 90.000,E1 140.598} C_DIS
LIN {X -0.250,Y -553.872,Z 1351.572,A 0.000,B 0.000,C 90.000,E1 138.933} C_DIS
LIN {X 0.030,Y -554.841,Z 1351.563,A 0.000,B 0.000,C 90.000,E1 137.229} C_DIS
LIN {X -0.170,Y -555.371,Z 1351.556,A 0.000,B 0.000,C 90.000,E1 136.134} C_DIS
LIN {X -0.217,Y -556.610,Z 1351.545,A 0.000,B 0.000,C 90.000,E1 134.190} C_DIS
LIN {X -0.042,Y -557.150,Z 1351.543,A 0.000,B 0.000,C 90.000,E1 133.785} C_DIS
LIN {X -0.083,Y -557.175,Z 1351.543,A 0.000,B 0.000,C 90.000,E1 133.785} C_DIS
LIN {X -0.115,Y -558.111,Z 1351.542,A 0.000,B 0.000,C 90.000,E1 133.623} C_DIS
LIN {X 0.010,Y -558.937,Z 1351.541,A 0.000,B 0.000,C 90.000,E1 133.380} C_DIS
LIN {X -0.032,Y -558.992,Z 1351.541,A 0.000,B 0.000,C 90.000,E1 133.380} C_DIS
LIN {X 0.005,Y -560.951,Z 1351.540,A 0.000,B 0.000,C 90.000,E1 133.218} C_DIS
LIN {X 0.084,Y -563.381,Z 1351.540,A 0.000,B 0.000,C 90.000,E1 133.095} C_DIS
LIN {X 0.009,Y -572.899,Z 1351.538,A 0.000,B 0.000,C 90.000,E1 132.852} C_DIS
LIN {X 0.192,Y -578.805,Z 1351.537,A 0.000,B 0.000,C 90.000,E1 132.609} C_DIS
LIN {X -0.326,Y -581.683,Z 1351.536,A 0.000,B 0.000,C 90.000,E1 132.528} C_DIS
LIN {X -0.243,Y -584.448,Z 1351.535,A 0.000,B 0.000,C 90.000,E1 132.366} C_DIS
LIN {X -0.271,Y -590.300,Z 1351.533,A 0.000,B 0.000,C 90.000,E1 132.000} C_DIS
LIN {X 0.073,Y -596.027,Z 1351.531,A 0.000,B 0.000,C 90.000,E1 131.553} C_DIS
LIN {X -0.349,Y -601.511,Z 1351.528,A 0.000,B 0.000,C 90.000,E1 131.148} C_DIS
LIN {X -0.172,Y -607.944,Z 1351.525,A 0.000,B 0.000,C 90.000,E1 130.539} C_DIS
LIN {X -0.167,Y -611.746,Z 1351.523,A 0.000,B 0.000,C 90.000,E1 130.172} C_DIS
LIN {X 0.099,Y -616.631,Z 1351.520,A 0.000,B 0.000,C 90.000,E1 129.644} C_DIS
LIN {X 0.212,Y -622.526,Z 1351.517,A 0.000,B 0.000,C 90.000,E1 128.991} C_DIS
LIN {X -0.127,Y -628.087,Z 1351.513,A 0.000,B 0.000,C 90.000,E1 128.382} C_DIS
LIN {X -0.307,Y -632.346,Z 1351.510,A 0.000,B 0.000,C 90.000,E1 127.890} C_DIS
LIN {X 0.009,Y -636.328,Z 1351.508,A 0.000,B 0.000,C 90.000,E1 127.363} C_DIS
LIN {X 0.133,Y -643.713,Z 1351.502,A 0.000,B 0.000,C 90.000,E1 126.377} C_DIS
LIN {X -0.009,Y -650.141,Z 1351.497,A 0.000,B 0.000,C 90.000,E1 125.518} C_DIS
LIN {X 0.036,Y -655.093,Z 1351.493,A 0.000,B 0.000,C 90.000,E1 124.771} C_DIS
LIN {X 0.028,Y -657.420,Z 1351.491,A 0.000,B 0.000,C 90.000,E1 124.405} C_DIS
LIN {X 0.046,Y -660.363,Z 1351.489,A 0.000,B 0.000,C 90.000,E1 123.913} C_DIS
LIN {X 0.139,Y -663.621,Z 1351.485,A 0.000,B 0.000,C 90.000,E1 123.293} C_DIS
LIN {X 0.257,Y -666.567,Z 1351.482,A 0.000,B 0.000,C 90.000,E1 122.673} C_DIS
LIN {X 0.111,Y -669.546,Z 1351.478,A 0.000,B 0.000,C 90.000,E1 121.957} C_DIS
LIN {X 0.196,Y -671.373,Z 1351.475,A 0.000,B 0.000,C 90.000,E1 121.465} C_DIS
LIN {X -0.304,Y -674.414,Z 1351.470,A 0.000,B 0.000,C 90.000,E1 120.541} C_DIS
LIN {X -0.023,Y -676.257,Z 1351.466,A 0.000,B 0.000,C 90.000,E1 119.795} C_DIS
LIN {X -0.248,Y -677.252,Z 1351.463,A 0.000,B 0.000,C 90.000,E1 119.333} C_DIS
LIN {X 0.127,Y -677.999,Z 1351.460,A 0.000,B 0.000,C 90.000,E1 118.821} C_DIS
LIN {X -0.085,Y -678.436,Z 1351.458,A 0.000,B 0.000,C 90.000,E1 118.359} C_DIS
LIN {X -0.102,Y -678.732,Z 1351.454,A 0.000,B 0.000,C 90.000,E1 117.641} C_DIS
LIN {X 0.074,Y -678.668,Z 1351.448,A 0.000,B 0.000,C 90.000,E1 116.668} C_DIS
LIN {X -0.248,Y -678.339,Z 1351.444,A 0.000,B 0.000,C 90.000,E1 115.976} C_DIS
LIN {X 0.334,Y -677.749,Z 1351.440,A 0.000,B 0.000,C 90.000,E1 115.207} C_DIS
LIN {X -0.183,Y -677.117,Z 1351.438,A 0.000,B 0.000,C 90.000,E1 114.771} C_DIS
LIN {X 0.006,Y -676.678,Z 1351.436,A 0.000,B 0.000,C 90.000,E1 114.515} C_DIS
LIN {X 0.194,Y -675.956,Z 1351.435,A 0.000,B 0.000,C 90.000,E1 114.259} C_DIS
LIN {X 0.286,Y -674.231,Z 1351.432,A 0.000,B 0.000,C 90.000,E1 113.770} C_DIS
LIN {X -0.065,Y -671.642,Z 1351.430,A 0.000,B 0.000,C 90.000,E1 113.439} C_DIS
LIN {X -0.162,Y -669.830,Z 1351.429,A 0.000,B 0.000,C 90.000,E1 113.206} C_DIS
LIN {X -0.080,Y -668.430,Z 1351.428,A 0.000,B 0.000,C 90.000,E1 113.078} C_DIS
LIN {X -0.053,Y -662.666,Z 1351.426,A 0.000,B 0.000,C 90.000,E1 112.695} C_DIS
LIN {X 0.027,Y -660.779,Z 1351.426,A 0.000,B 0.000,C 90.000,E1 112.589} C_DIS
LIN {X -0.113,Y -654.367,Z 1351.424,A 0.000,B 0.000,C 90.000,E1 112.386} C_DIS
LIN {X -0.213,Y -649.479,Z 1351.424,A 0.000,B 0.000,C 90.000,E1 112.280} C_DIS
LIN {X 0.214,Y -637.183,Z 1351.422,A 0.000,B 0.000,C 90.000,E1 111.972} C_DIS
LIN {X -0.052,Y -636.333,Z 1351.422,A 0.000,B 0.000,C 90.000,E1 111.972} C_DIS
LIN {X -0.105,Y -636.246,Z 1351.422,A 0.000,B 0.000,C 90.000,E1 111.972} C_DIS
LIN {X -0.192,Y -637.027,Z 1351.421,A 0.000,B 0.000,C 90.000,E1 111.844} C_DIS
LIN {X 0.229,Y -645.572,Z 1351.416,A 0.000,B 0.000,C 90.000,E1 110.791} C_DIS
LIN {X 0.170,Y -650.278,Z 1351.412,A 0.000,B 0.000,C 90.000,E1 110.174} C_DIS
LIN {X -0.034,Y -654.706,Z 1351.408,A 0.000,B 0.000,C 90.000,E1 109.450} C_DIS
LIN {X -0.242,Y -657.821,Z 1351.405,A 0.000,B 0.000,C 90.000,E1 108.852} C_DIS
LIN {X -0.168,Y -661.125,Z 1351.401,A 0.000,B 0.000,C 90.000,E1 108.109} C_DIS
LIN {X 0.170,Y -666.022,Z 1351.394,A 0.000,B 0.000,C 90.000,E1 106.858} C_DIS
LIN {X 0.109,Y -668.523,Z 1351.390,A 0.000,B 0.000,C 90.000,E1 106.134} C_DIS
LIN {X -0.044,Y -669.971,Z 1351.387,A 0.000,B 0.000,C 90.000,E1 105.662} C_DIS
LIN {X -0.253,Y -671.747,Z 1351.383,A 0.000,B 0.000,C 90.000,E1 104.954} C_DIS
LIN {X -0.379,Y -672.805,Z 1351.380,A 0.000,B 0.000,C 90.000,E1 104.481} C_DIS
LIN {X 0.098,Y -673.917,Z 1351.376,A 0.000,B 0.000,C 90.000,E1 103.716} C_DIS
LIN {X -0.013,Y -674.389,Z 1351.374,A 0.000,B 0.000,C 90.000,E1 103.244} C_DIS
LIN {X -0.176,Y -674.751,Z 1351.370,A 0.000,B 0.000,C 90.000,E1 102.535} C_DIS
LIN {X -0.284,Y -674.738,Z 1351.367,A 0.000,B 0.000,C 90.000,E1 102.063} C_DIS
LIN {X 0.265,Y -674.534,Z 1351.364,A 0.000,B 0.000,C 90.000,E1 101.535} C_DIS
LIN {X -0.039,Y -673.866,Z 1351.360,A 0.000,B 0.000,C 90.000,E1 100.838} C_DIS
LIN {X -0.160,Y -673.211,Z 1351.358,A 0.000,B 0.000,C 90.000,E1 100.366} C_DIS
LIN {X 0.256,Y -672.278,Z 1351.355,A 0.000,B 0.000,C 90.000,E1 99.849} C_DIS
LIN {X 0.118,Y -671.035,Z 1351.352,A 0.000,B 0.000,C 90.000,E1 99.378} C_DIS
LIN {X -0.216,Y -668.677,Z 1351.348,A 0.000,B 0.000,C 90.000,E1 98.681} C_DIS
LIN {X 0.176,Y -666.860,Z 1351.345,A 0.000,B 0.000,C 90.000,E1 98.163} C_DIS
LIN {X -0.100,Y -664.834,Z 1351.343,A 0.000,B 0.000,C 90.000,E1 97.701} C_DIS
LIN {X 0.176,Y -661.970,Z 1351.339,A 0.000,B 0.000,C 90.000,E1 97.068} C_DIS
LIN {X 0.173,Y -656.183,Z 1351.333,A 0.000,B 0.000,C 90.000,E1 95.967} C_DIS
LIN {X -0.238,Y -653.385,Z 1351.331,A 0.000,B 0.000,C 90.000,E1 95.511} C_DIS
LIN {X -0.220,Y -647.934,Z 1351.326,A 0.000,B 0.000,C 90.000,E1 94.645} C_DIS
LIN {X -0.090,Y -643.647,Z 1351.322,A 0.000,B 0.000,C 90.000,E1 94.012} C_DIS
LIN {X -0.039,Y -638.944,Z 1351.319,A 0.000,B 0.000,C 90.000,E1 93.383} C_DIS
LIN {X 0.012,Y -633.231,Z 1351.315,A 0.000,B 0.000,C 90.000,E1 92.751} C_DIS
LIN {X -0.140,Y -623.255,Z 1351.310,A 0.000,B 0.000,C 90.000,E1 91.776} C_DIS
LIN {X 0.042,Y -616.904,Z 1351.306,A 0.000,B 0.000,C 90.000,E1 91.146} C_DIS
LIN {X -0.144,Y -610.086,Z 1351.303,A 0.000,B 0.000,C 90.000,E1 90.573} C_DIS
LIN {X -0.042,Y -605.208,Z 1351.301,A 0.000,B 0.000,C 90.000,E1 90.229} C_DIS
LIN {X 0.266,Y -602.175,Z 1351.300,A 0.000,B 0.000,C 90.000,E1 90.000} C_DIS
LIN {X 0.128,Y -595.429,Z 1351.298,A 0.000,B 0.000,C 90.000,E1 89.656} C_DIS
LIN {X -0.153,Y -586.559,Z 1351.296,A 0.000,B 0.000,C 90.000,E1 89.312} C_DIS
LIN {X -0.029,Y -580.198,Z 1351.295,A 0.000,B 0.000,C 90.000,E1 89.026} C_DIS
LIN {X -0.268,Y -577.339,Z 1351.294,A 0.000,B 0.000,C 90.000,E1 88.912} C_DIS
LIN {X 0.158,Y -574.777,Z 1351.293,A 0.000,B 0.000,C 90.000,E1 88.682} C_DIS
LIN {X -0.286,Y -573.411,Z 1351.292,A 0.000,B 0.000,C 90.000,E1 88.568} C_DIS
LIN {X 0.005,Y -573.214,Z 1351.292,A 0.000,B 0.000,C 90.000,E1 88.511} C_DIS
LIN {X -0.031,Y -573.193,Z 1351.292,A 0.000,B 0.000,C 90.000,E1 88.511} C_DIS
LIN {X -0.139,Y -572.773,Z 1351.290,A 0.000,B 0.000,C 90.000,E1 88.224} C_DIS
LIN {X -0.193,Y -573.188,Z 1351.286,A 0.000,B 0.000,C 90.000,E1 87.535} C_DIS
LIN {X 0.279,Y -574.981,Z 1351.276,A 0.000,B 0.000,C 90.000,E1 85.584} C_DIS
LIN {X -0.105,Y -577.400,Z 1351.264,A 0.000,B 0.000,C 90.000,E1 83.451} C_DIS
LIN {X -0.210,Y -579.284,Z 1351.255,A 0.000,B 0.000,C 90.000,E1 81.837} C_DIS
LIN {X -0.110,Y -581.256,Z 1351.246,A 0.000,B 0.000,C 90.000,E1 80.208} C_DIS
LIN {X -0.199,Y -582.697,Z 1351.238,A 0.000,B 0.000,C 90.000,E1 78.870} C_DIS
LIN {X -0.153,Y -584.024,Z 1351.231,A 0.000,B 0.000,C 90.000,E1 77.521} C_DIS
LIN {X -0.086,Y -585.172,Z 1351.223,A 0.000,B 0.000,C 90.000,E1 76.172} C_DIS
LIN {X 0.138,Y -586.255,Z 1351.216,A 0.000,B 0.000,C 90.000,E1 74.810} C_DIS
LIN {X -0.190,Y -587.130,Z 1351.208,A 0.000,B 0.000,C 90.000,E1 73.504} C_DIS
LIN {X 0.081,Y -588.123,Z 1351.199,A 0.000,B 0.000,C 90.000,E1 71.873} C_DIS
LIN {X -0.177,Y -589.070,Z 1351.190,A 0.000,B 0.000,C 90.000,E1 70.296} C_DIS
LIN {X -0.094,Y -589.862,Z 1351.183,A 0.000,B 0.000,C 90.000,E1 68.954} C_DIS
LIN {X -0.120,Y -590.916,Z 1351.174,A 0.000,B 0.000,C 90.000,E1 67.358} C_DIS
LIN {X -0.008,Y -592.342,Z 1351.164,A 0.000,B 0.000,C 90.000,E1 65.485} C_DIS
LIN {X 0.134,Y -593.164,Z 1351.158,A 0.000,B 0.000,C 90.000,E1 64.409} C_DIS
LIN {X 0.096,Y -594.245,Z 1351.149,A 0.000,B 0.000,C 90.000,E1 62.820} C_DIS
LIN {X -0.070,Y -595.991,Z 1351.137,A 0.000,B 0.000,C 90.000,E1 60.717} C_DIS
LIN {X -0.184,Y -598.136,Z 1351.126,A 0.000,B 0.000,C 90.000,E1 58.614} C_DIS
LIN {X -0.280,Y -599.647,Z 1351.117,A 0.000,B 0.000,C 90.000,E1 57.041} C_DIS
LIN {X 0.010,Y -600.690,Z 1351.111,A 0.000,B 0.000,C 90.000,E1 55.960} C_DIS
LIN {X -0.188,Y -602.192,Z 1351.102,A 0.000,B 0.000,C 90.000,E1 54.402} C_DIS
LIN {X -0.092,Y -603.913,Z 1351.092,A 0.000,B 0.000,C 90.000,E1 52.557} C_DIS
LIN {X 0.093,Y -604.684,Z 1351.086,A 0.000,B 0.000,C 90.000,E1 51.492} C_DIS
LIN {X 0.246,Y -605.664,Z 1351.077,A 0.000,B 0.000,C 90.000,E1 49.908} C_DIS
LIN {X 0.367,Y -606.160,Z 1351.072,A 0.000,B 0.000,C 90.000,E1 48.852} C_DIS
LIN {X 0.233,Y -606.436,Z 1351.067,A 0.000,B 0.000,C 90.000,E1 48.081} C_DIS
LIN {X 0.164,Y -606.754,Z 1351.060,A 0.000,B 0.000,C 90.000,E1 46.782} C_DIS
LIN {X -0.118,Y -606.914,Z 1351.051,A 0.000,B 0.000,C 90.000,E1 45.243} C_DIS
LIN {X -0.015,Y -606.783,Z 1351.046,A 0.000,B 0.000,C 90.000,E1 44.190} C_DIS
LIN {X 0.081,Y -606.423,Z 1351.040,A 0.000,B 0.000,C 90.000,E1 43.137} C_DIS
LIN {X -0.189,Y -605.745,Z 1351.031,A 0.000,B 0.000,C 90.000,E1 41.595} C_DIS
LIN {X 0.188,Y -605.017,Z 1351.024,A 0.000,B 0.000,C 90.000,E1 40.253} C_DIS
LIN {X 0.085,Y -604.325,Z 1351.016,A 0.000,B 0.000,C 90.000,E1 38.955} C_DIS
LIN {X 0.053,Y -603.445,Z 1351.009,A 0.000,B 0.000,C 90.000,E1 37.649} C_DIS
LIN {X 0.233,Y -602.416,Z 1351.003,A 0.000,B 0.000,C 90.000,E1 36.583} C_DIS
LIN {X 0.151,Y -601.355,Z 1350.999,A 0.000,B 0.000,C 90.000,E1 35.804} C_DIS
LIN {X 0.058,Y -600.069,Z 1350.995,A 0.000,B 0.000,C 90.000,E1 35.025} C_DIS
LIN {X 0.082,Y -597.437,Z 1350.987,A 0.000,B 0.000,C 90.000,E1 33.706} C_DIS
LIN {X 0.112,Y -595.655,Z 1350.983,A 0.000,B 0.000,C 90.000,E1 32.911} C_DIS
LIN {X -0.154,Y -592.943,Z 1350.977,A 0.000,B 0.000,C 90.000,E1 31.878} C_DIS
LIN {X -0.052,Y -591.342,Z 1350.974,A 0.000,B 0.000,C 90.000,E1 31.337} C_DIS
LIN {X 0.113,Y -587.772,Z 1350.968,A 0.000,B 0.000,C 90.000,E1 30.256} C_DIS
LIN {X -0.119,Y -585.852,Z 1350.965,A 0.000,B 0.000,C 90.000,E1 29.745} C_DIS
LIN {X -0.071,Y -583.690,Z 1350.962,A 0.000,B 0.000,C 90.000,E1 29.205} C_DIS
LIN {X 0.197,Y -578.831,Z 1350.956,A 0.000,B 0.000,C 90.000,E1 28.103} C_DIS
LIN {X -0.047,Y -573.946,Z 1350.951,A 0.000,B 0.000,C 90.000,E1 27.180} C_DIS
LIN {X 0.066,Y -570.226,Z 1350.947,A 0.000,B 0.000,C 90.000,E1 26.488} C_DIS
LIN {X 0.149,Y -566.095,Z 1350.943,A 0.000,B 0.000,C 90.000,E1 25.796} C_DIS
LIN {X 0.006,Y -559.819,Z 1350.938,A 0.000,B 0.000,C 90.000,E1 24.847} C_DIS
LIN {X -0.104,Y -553.782,Z 1350.933,A 0.000,B 0.000,C 90.000,E1 24.027} C_DIS
LIN {X -0.280,Y -547.379,Z 1350.929,A 0.000,B 0.000,C 90.000,E1 23.206} C_DIS
LIN {X -0.027,Y -540.288,Z 1350.924,A 0.000,B 0.000,C 90.000,E1 22.333} C_DIS
LIN {X 0.148,Y -532.815,Z 1350.919,A 0.000,B 0.000,C 90.000,E1 21.461} C_DIS
LIN {X 0.154,Y -523.834,Z 1350.914,A 0.000,B 0.000,C 90.000,E1 20.482} C_DIS
LIN {X 0.030,Y -512.043,Z 1350.907,A 0.000,B 0.000,C 90.000,E1 19.268} C_DIS
LIN {X 0.072,Y -504.228,Z 1350.902,A 0.000,B 0.000,C 90.000,E1 18.417} C_DIS
LIN {X 0.169,Y -493.151,Z 1350.896,A 0.000,B 0.000,C 90.000,E1 17.275} C_DIS
LIN {X -0.172,Y -484.410,Z 1350.892,A 0.000,B 0.000,C 90.000,E1 16.496} C_DIS
LIN {X 0.147,Y -467.424,Z 1350.883,A 0.000,B 0.000,C 90.000,E1 14.828} C_DIS
LIN {X -0.250,Y -456.059,Z 1350.876,A 0.000,B 0.000,C 90.000,E1 13.772} C_DIS
LIN {X -0.033,Y -436.099,Z 1350.865,A 0.000,B 0.000,C 90.000,E1 11.715} C_DIS
LIN {X 0.127,Y -419.201,Z 1350.855,A 0.000,B 0.000,C 90.000,E1 9.849} C_DIS
LIN {X 0.158,Y -406.465,Z 1350.847,A 0.000,B 0.000,C 90.000,E1 8.398} C_DIS
LIN {X -0.162,Y -398.049,Z 1350.841,A 0.000,B 0.000,C 90.000,E1 7.466} C_DIS
LIN {X -0.144,Y -396.674,Z 1350.840,A 0.000,B 0.000,C 90.000,E1 7.296} C_DIS
LIN {X -0.117,Y -394.212,Z 1350.838,A 0.000,B 0.000,C 90.000,E1 6.891} C_DIS
LIN {X -0.154,Y -394.197,Z 1350.838,A 0.000,B 0.000,C 90.000,E1 6.891} C_DIS
LIN {X -0.131,Y -394.850,Z 1350.838,A 0.000,B 0.000,C 90.000,E1 6.777} C_DIS
LIN {X 0.046,Y -395.562,Z 1350.837,A 0.000,B 0.000,C 90.000,E1 6.663} C_DIS
LIN {X -0.082,Y -399.749,Z 1350.835,A 0.000,B 0.000,C 90.000,E1 6.315} C_DIS
LIN {X 0.148,Y -412.287,Z 1350.830,A 0.000,B 0.000,C 90.000,E1 5.391} C_DIS
LIN {X 0.068,Y -417.163,Z 1350.828,A 0.000,B 0.000,C 90.000,E1 5.049} C_DIS
LIN {X 0.107,Y -423.198,Z 1350.825,A 0.000,B 0.000,C 90.000,E1 4.531} C_DIS
LIN {X 0.008,Y -430.406,Z 1350.821,A 0.000,B 0.000,C 90.000,E1 3.841} C_DIS
LIN {X 0.004,Y -437.376,Z 1350.817,A 0.000,B 0.000,C 90.000,E1 3.094} C_DIS
LIN {X 0.139,Y -444.147,Z 1350.813,A 0.000,B 0.000,C 90.000,E1 2.293} C_DIS
LIN {X -0.042,Y -449.229,Z 1350.810,A 0.000,B 0.000,C 90.000,E1 1.718} C_DIS
LIN {X -0.100,Y -455.573,Z 1350.805,A 0.000,B 0.000,C 90.000,E1 0.917} C_DIS
LIN {X -0.098,Y -461.480,Z 1350.801,A 0.000,B 0.000,C 90.000,E1 0.115} C_DIS
LIN {X 0.034,Y -466.862,Z 1350.796,A 0.000,B 0.000,C 90.000,E1 359.312} C_DIS
LIN {X 0.146,Y -471.922,Z 1350.792,A 0.000,B 0.000,C 90.000,E1 358.511} C_DIS
LIN {X -0.018,Y -477.401,Z 1350.787,A 0.000,B 0.000,C 90.000,E1 357.593} C_DIS
LIN {X 0.052,Y -480.891,Z 1350.783,A 0.000,B 0.000,C 90.000,E1 356.963} C_DIS
LIN {X -0.161,Y -484.924,Z 1350.779,A 0.000,B 0.000,C 90.000,E1 356.216} C_DIS
LIN {X 0.149,Y -488.563,Z 1350.775,A 0.000,B 0.000,C 90.000,E1 355.412} C_DIS
LIN {X -0.155,Y -491.256,Z 1350.771,A 0.000,B 0.000,C 90.000,E1 354.837} C_DIS
LIN {X 0.052,Y -493.802,Z 1350.768,A 0.000,B 0.000,C 90.000,E1 354.204} C_DIS
LIN {X 0.178,Y -497.291,Z 1350.763,A 0.000,B 0.000,C 90.000,E1 353.280} C_DIS
LIN {X -0.153,Y -500.423,Z 1350.758,A 0.000,B 0.000,C 90.000,E1 352.413} C_DIS
LIN {X 0.264,Y -501.439,Z 1350.756,A 0.000,B 0.000,C 90.000,E1 352.064} C_DIS
LIN {X -0.087,Y -504.858,Z 1350.750,A 0.000,B 0.000,C 90.000,E1 350.905} C_DIS
LIN {X 0.157,Y -507.170,Z 1350.745,A 0.000,B 0.000,C 90.000,E1 349.982} C_DIS
LIN {X 0.011,Y -509.219,Z 1350.740,A 0.000,B 0.000,C 90.000,E1 349.106} C_DIS
LIN {X -0.111,Y -511.108,Z 1350.735,A 0.000,B 0.000,C 90.000,E1 348.229} C_DIS
LIN {X -0.214,Y -512.804,Z 1350.730,A 0.000,B 0.000,C 90.000,E1 347.353} C_DIS
LIN {X -0.184,Y -514.227,Z 1350.725,A 0.000,B 0.000,C 90.000,E1 346.464} C_DIS
LIN {X -0.156,Y -515.873,Z 1350.718,A 0.000,B 0.000,C 90.000,E1 345.283} C_DIS
LIN {X -0.108,Y -517.064,Z 1350.712,A 0.000,B 0.000,C 90.000,E1 344.102} C_DIS
LIN {X 0.117,Y -517.655,Z 1350.707,A 0.000,B 0.000,C 90.000,E1 343.196} C_DIS
LIN {X 0.199,Y -518.015,Z 1350.702,A 0.000,B 0.000,C 90.000,E1 342.308} C_DIS
LIN {X -0.053,Y -518.074,Z 1350.697,A 0.000,B 0.000,C 90.000,E1 341.456} C_DIS
LIN {X 0.188,Y -517.888,Z 1350.692,A 0.000,B 0.000,C 90.000,E1 340.550} C_DIS
LIN {X -0.200,Y -517.577,Z 1350.689,A 0.000,B 0.000,C 90.000,E1 340.007} C_DIS
LIN {X -0.062,Y -517.238,Z 1350.687,A 0.000,B 0.000,C 90.000,E1 339.699} C_DIS
LIN {X 0.074,Y -516.740,Z 1350.686,A 0.000,B 0.000,C 90.000,E1 339.390} C_DIS
LIN {X 0.211,Y -516.040,Z 1350.684,A 0.000,B 0.000,C 90.000,E1 339.082} C_DIS
LIN {X -0.135,Y -515.069,Z 1350.682,A 0.000,B 0.000,C 90.000,E1 338.827} C_DIS
LIN {X 0.171,Y -514.426,Z 1350.682,A 0.000,B 0.000,C 90.000,E1 338.646} C_DIS
LIN {X -0.190,Y -513.559,Z 1350.681,A 0.000,B 0.000,C 90.000,E1 338.539} C_DIS
LIN {X 0.110,Y -512.202,Z 1350.680,A 0.000,B 0.000,C 90.000,E1 338.358} C_DIS
LIN {X 0.087,Y -505.481,Z 1350.678,A 0.000,B 0.000,C 90.000,E1 338.050} C_DIS
LIN {X -0.047,Y -475.216,Z 1350.670,A 0.000,B 0.000,C 90.000,E1 336.613} C_DIS
LIN {X 0.012,Y -448.573,Z 1350.662,A 0.000,B 0.000,C 90.000,E1 335.153} C_DIS
LIN {X -0.069,Y -423.900,Z 1350.654,A 0.000,B 0.000,C 90.000,E1 333.640} C_DIS
LIN {X 0.139,Y -401.199,Z 1350.645,A 0.000,B 0.000,C 90.000,E1 332.025} C_DIS
LIN {X -0.012,Y -380.449,Z 1350.636,A 0.000,B 0.000,C 90.000,E1 330.411} C_DIS
LIN {X -0.135,Y -367.263,Z 1350.629,A 0.000,B 0.000,C 90.000,E1 329.282} C_DIS
LIN {X 0.024,Y -367.252,Z 1350.629,A 0.000,B 0.000,C 90.000,E1 329.253} C_DIS
LIN {X 0.194,Y -371.793,Z 1350.601,A 0.000,B 0.000,C 90.000,E1 324.196} C_DIS
LIN {X -0.017,Y -377.413,Z 1350.567,A 0.000,B 0.000,C 90.000,E1 318.000} C_DIS
LIN {X 0.007,Y -378.261,Z 1350.563,A 0.000,B 0.000,C 90.000,E1 317.268} C_DIS
LIN {X 0.005,Y -383.997,Z 1350.530,A 0.000,B 0.000,C 90.000,E1 311.472} C_DIS
LIN {X 0.055,Y -384.920,Z 1350.526,A 0.000,B 0.000,C 90.000,E1 310.744} C_DIS
LIN {X -0.025,Y -390.667,Z 1350.495,A 0.000,B 0.000,C 90.000,E1 305.025} C_DIS
LIN {X -0.181,Y -391.164,Z 1350.493,A 0.000,B 0.000,C 90.000,E1 304.692} C_DIS
LIN {X -0.092,Y -392.715,Z 1350.481,A 0.000,B 0.000,C 90.000,E1 302.546} C_DIS
LIN {X 0.171,Y -396.881,Z 1350.459,A 0.000,B 0.000,C 90.000,E1 298.615} C_DIS
LIN {X 0.075,Y -397.304,Z 1350.455,A 0.000,B 0.000,C 90.000,E1 297.924} C_DIS
LIN {X 0.182,Y -401.627,Z 1350.426,A 0.000,B 0.000,C 90.000,E1 292.642} C_DIS
LIN {X -0.067,Y -404.696,Z 1350.395,A 0.000,B 0.000,C 90.000,E1 287.094} C_DIS
LIN {X -0.075,Y -404.825,Z 1350.383,A 0.000,B 0.000,C 90.000,E1 285.009} C_DIS
LIN {X -0.076,Y -406.124,Z 1350.364,A 0.000,B 0.000,C 90.000,E1 281.535} C_DIS
LIN {X -0.044,Y -405.828,Z 1350.358,A 0.000,B 0.000,C 90.000,E1 280.489} C_DIS
LIN {X 0.016,Y -405.688,Z 1350.333,A 0.000,B 0.000,C 90.000,E1 275.967} C_DIS
LIN {X 0.054,Y -403.471,Z 1350.304,A 0.000,B 0.000,C 90.000,E1 270.745} C_DIS
LIN {X 0.022,Y -403.259,Z 1350.302,A 0.000,B 0.000,C 90.000,E1 270.401} C_DIS
LIN {X -0.196,Y -398.883,Z 1350.271,A 0.000,B 0.000,C 90.000,E1 264.837} C_DIS
LIN {X 0.098,Y -393.354,Z 1350.244,A 0.000,B 0.000,C 90.000,E1 259.859} C_DIS
LIN {X 0.020,Y -392.786,Z 1350.240,A 0.000,B 0.000,C 90.000,E1 259.162} C_DIS
LIN {X 0.098,Y -386.334,Z 1350.214,A 0.000,B 0.000,C 90.000,E1 254.519} C_DIS
LIN {X 0.059,Y -385.227,Z 1350.208,A 0.000,B 0.000,C 90.000,E1 253.449} C_DIS
LIN {X 0.100,Y -384.033,Z 1350.204,A 0.000,B 0.000,C 90.000,E1 252.725} C_DIS
LIN {X -0.071,Y -377.460,Z 1350.180,A 0.000,B 0.000,C 90.000,E1 248.411} C_DIS
LIN {X 0.021,Y -376.186,Z 1350.174,A 0.000,B 0.000,C 90.000,E1 247.305} C_DIS
LIN {X 0.037,Y -369.930,Z 1350.154,A 0.000,B 0.000,C 90.000,E1 243.640} C_DIS
LIN {X 0.052,Y -366.493,Z 1350.139,A 0.000,B 0.000,C 90.000,E1 241.051} C_DIS
LIN {X 0.137,Y -365.962,Z 1350.137,A 0.000,B 0.000,C 90.000,E1 240.667} C_DIS
LIN {X 0.027,Y -359.134,Z 1350.114,A 0.000,B 0.000,C 90.000,E1 236.580} C_DIS
LIN {X 0.022,Y -356.273,Z 1350.102,A 0.000,B 0.000,C 90.000,E1 234.322} C_DIS
LIN {X 0.242,Y -355.761,Z 1350.100,A 0.000,B 0.000,C 90.000,E1 233.909} C_DIS
LIN {X 0.045,Y -348.737,Z 1350.074,A 0.000,B 0.000,C 90.000,E1 229.380} C_DIS
LIN {X 0.119,Y -346.140,Z 1350.062,A 0.000,B 0.000,C 90.000,E1 227.067} C_DIS
LIN {X 0.007,Y -344.395,Z 1350.055,A 0.000,B 0.000,C 90.000,E1 225.931} C_DIS
LIN {X -0.092,Y -338.163,Z 1350.027,A 0.000,B 0.000,C 90.000,E1 220.906} C_DIS
LIN {X 0.036,Y -336.786,Z 1350.019,A 0.000,B 0.000,C 90.000,E1 219.322} C_DIS
LIN {X -0.146,Y -331.635,Z 1349.993,A 0.000,B 0.000,C 90.000,E1 214.818} C_DIS
LIN {X -0.163,Y -331.656,Z 1349.993,A 0.000,B 0.000,C 90.000,E1 214.818} C_DIS
LIN {X 0.042,Y -348.755,Z 1349.983,A 0.000,B 0.000,C 90.000,E1 212.911} C_DIS
LIN {X 0.124,Y -367.792,Z 1349.973,A 0.000,B 0.000,C 90.000,E1 211.052} C_DIS
LIN {X -0.044,Y -387.173,Z 1349.963,A 0.000,B 0.000,C 90.000,E1 209.411} C_DIS
LIN {X 0.040,Y -408.494,Z 1349.954,A 0.000,B 0.000,C 90.000,E1 207.769} C_DIS
LIN {X 0.126,Y -431.790,Z 1349.946,A 0.000,B 0.000,C 90.000,E1 206.181} C_DIS
LIN {X -0.118,Y -446.918,Z 1349.940,A 0.000,B 0.000,C 90.000,E1 205.283} C_DIS
LIN {X -0.082,Y -448.723,Z 1349.939,A 0.000,B 0.000,C 90.000,E1 205.079} C_DIS
LIN {X -0.088,Y -450.288,Z 1349.938,A 0.000,B 0.000,C 90.000,E1 204.771} C_DIS
LIN {X -0.215,Y -451.465,Z 1349.936,A 0.000,B 0.000,C 90.000,E1 204.463} C_DIS
LIN {X -0.147,Y -452.408,Z 1349.934,A 0.000,B 0.000,C 90.000,E1 204.131} C_DIS
LIN {X 0.151,Y -453.156,Z 1349.932,A 0.000,B 0.000,C 90.000,E1 203.770} C_DIS
LIN {X 0.113,Y -454.249,Z 1349.929,A 0.000,B 0.000,C 90.000,E1 203.131} C_DIS
LIN {X 0.025,Y -456.126,Z 1349.920,A 0.000,B 0.000,C 90.000,E1 201.535} C_DIS
LIN {X 0.072,Y -457.536,Z 1349.913,A 0.000,B 0.000,C 90.000,E1 200.248} C_DIS
LIN {X 0.066,Y -460.315,Z 1349.898,A 0.000,B 0.000,C 90.000,E1 197.692} C_DIS
LIN {X -0.071,Y -462.364,Z 1349.886,A 0.000,B 0.000,C 90.000,E1 195.481} C_DIS
LIN {X 0.059,Y -464.301,Z 1349.874,A 0.000,B 0.000,C 90.000,E1 193.244} C_DIS
LIN {X 0.242,Y -466.359,Z 1349.861,A 0.000,B 0.000,C 90.000,E1 191.007} C_DIS
LIN {X -0.149,Y -467.449,Z 1349.854,A 0.000,B 0.000,C 90.000,E1 189.792} C_DIS
LIN {X 0.019,Y -468.540,Z 1349.847,A 0.000,B 0.000,C 90.000,E1 188.511} C_DIS
LIN {X 0.132,Y -469.406,Z 1349.840,A 0.000,B 0.000,C 90.000,E1 187.239} C_DIS
LIN {X 0.015,Y -470.201,Z 1349.832,A 0.000,B 0.000,C 90.000,E1 185.682} C_DIS
LIN {X -0.130,Y -470.747,Z 1349.823,A 0.000,B 0.000,C 90.000,E1 184.131} C_DIS
LIN {X 0.160,Y -470.905,Z 1349.818,A 0.000,B 0.000,C 90.000,E1 183.154} C_DIS
LIN {X 0.228,Y -470.860,Z 1349.811,A 0.000,B 0.000,C 90.000,E1 181.892} C_DIS
LIN {X 0.040,Y -470.577,Z 1349.806,A 0.000,B 0.000,C 90.000,E1 180.974} C_DIS
LIN {X -0.161,Y -470.048,Z 1349.800,A 0.000,B 0.000,C 90.000,E1 180.057} C_DIS
LIN {X -0.141,Y -469.544,Z 1349.797,A 0.000,B 0.000,C 90.000,E1 179.427} C_DIS
LIN {X 0.114,Y -468.545,Z 1349.792,A 0.000,B 0.000,C 90.000,E1 178.453} C_DIS
LIN {X -0.098,Y -467.402,Z 1349.786,A 0.000,B 0.000,C 90.000,E1 177.535} C_DIS
LIN {X 0.148,Y -465.960,Z 1349.781,A 0.000,B 0.000,C 90.000,E1 176.560} C_DIS
LIN {X 0.124,Y -463.595,Z 1349.774,A 0.000,B 0.000,C 90.000,E1 175.298} C_DIS
LIN {X -0.089,Y -462.919,Z 1349.772,A 0.000,B 0.000,C 90.000,E1 175.008} C_DIS
LIN {X -0.099,Y -461.182,Z 1349.769,A 0.000,B 0.000,C 90.000,E1 174.375} C_DIS
LIN {X 0.113,Y -457.992,Z 1349.763,A 0.000,B 0.000,C 90.000,E1 173.394} C_DIS
LIN {X -0.170,Y -453.806,Z 1349.758,A 0.000,B 0.000,C 90.000,E1 172.470} C_DIS
LIN {X 0.189,Y -450.625,Z 1349.755,A 0.000,B 0.000,C 90.000,E1 171.781} C_DIS
LIN {X 0.137,Y -447.119,Z 1349.751,A 0.000,B 0.000,C 90.000,E1 171.141} C_DIS
LIN {X 0.110,Y -442.062,Z 1349.746,A 0.000,B 0.000,C 90.000,E1 170.330} C_DIS
LIN {X 0.111,Y -436.457,Z 1349.742,A 0.000,B 0.000,C 90.000,E1 169.511} C_DIS
LIN {X 0.179,Y -428.509,Z 1349.735,A 0.000,B 0.000,C 90.000,E1 168.342} C_DIS
LIN {X -0.068,Y -415.274,Z 1349.724,A 0.000,B 0.000,C 90.000,E1 166.353} C_DIS
LIN {X 0.113,Y -410.816,Z 1349.720,A 0.000,B 0.000,C 90.000,E1 165.644} C_DIS
LIN {X -0.139,Y -406.974,Z 1349.717,A 0.000,B 0.000,C 90.000,E1 164.991} C_DIS
LIN {X -0.080,Y -406.136,Z 1349.716,A 0.000,B 0.000,C 90.000,E1 164.810} C_DIS
LIN {X -0.088,Y -403.928,Z 1349.712,A 0.000,B 0.000,C 90.000,E1 164.157} C_DIS
LIN {X -0.037,Y -403.462,Z 1349.711,A 0.000,B 0.000,C 90.000,E1 163.976} C_DIS
LIN {X 0.110,Y -403.482,Z 1349.709,A 0.000,B 0.000,C 90.000,E1 163.614} C_DIS
LIN {X 0.083,Y -403.504,Z 1349.709,A 0.000,B 0.000,C 90.000,E1 163.614} C_DIS
LIN {X -0.031,Y -405.048,Z 1349.708,A 0.000,B 0.000,C 90.000,E1 163.378} C_DIS
LIN {X 0.019,Y -405.920,Z 1349.707,A 0.000,B 0.000,C 90.000,E1 163.196} C_DIS
LIN {X 0.144,Y -410.260,Z 1349.704,A 0.000,B 0.000,C 90.000,E1 162.670} C_DIS
LIN {X -0.102,Y -417.027,Z 1349.700,A 0.000,B 0.000,C 90.000,E1 162.054} C_DIS
LIN {X 0.097,Y -422.671,Z 1349.698,A 0.000,B 0.000,C 90.000,E1 161.529} C_DIS
LIN {X 0.119,Y -444.533,Z 1349.688,A 0.000,B 0.000,C 90.000,E1 159.826} C_DIS
LIN {X -0.148,Y -457.216,Z 1349.683,A 0.000,B 0.000,C 90.000,E1 158.901} C_DIS
LIN {X -0.014,Y -466.463,Z 1349.679,A 0.000,B 0.000,C 90.000,E1 158.156} C_DIS
LIN {X -0.042,Y -474.002,Z 1349.675,A 0.000,B 0.000,C 90.000,E1 157.539} C_DIS
LIN {X -0.180,Y -481.501,Z 1349.672,A 0.000,B 0.000,C 90.000,E1 156.922} C_DIS
LIN {X 0.158,Y -490.046,Z 1349.667,A 0.000,B 0.000,C 90.000,E1 156.102} C_DIS
LIN {X -0.179,Y -494.261,Z 1349.665,A 0.000,B 0.000,C 90.000,E1 155.741} C_DIS
LIN {X -0.237,Y -502.476,Z 1349.661,A 0.000,B 0.000,C 90.000,E1 154.921} C_DIS
LIN {X -0.157,Y -509.064,Z 1349.657,A 0.000,B 0.000,C 90.000,E1 154.204} C_DIS
LIN {X 0.131,Y -514.139,Z 1349.653,A 0.000,B 0.000,C 90.000,E1 153.589} C_DIS
LIN {X -0.159,Y -517.813,Z 1349.651,A 0.000,B 0.000,C 90.000,E1 153.179} C_DIS
LIN {X 0.096,Y -522.245,Z 1349.648,A 0.000,B 0.000,C 90.000,E1 152.564} C_DIS
LIN {X 0.158,Y -526.247,Z 1349.644,A 0.000,B 0.000,C 90.000,E1 151.975} C_DIS
LIN {X 0.252,Y -529.853,Z 1349.641,A 0.000,B 0.000,C 90.000,E1 151.385} C_DIS
LIN {X 0.228,Y -533.559,Z 1349.637,A 0.000,B 0.000,C 90.000,E1 150.667} C_DIS
LIN {X -0.088,Y -536.014,Z 1349.634,A 0.000,B 0.000,C 90.000,E1 150.127} C_DIS
LIN {X 0.072,Y -539.140,Z 1349.629,A 0.000,B 0.000,C 90.000,E1 149.253} C_DIS
LIN {X -0.003,Y -542.671,Z 1349.623,A 0.000,B 0.000,C 90.000,E1 148.122} C_DIS
LIN {X 0.229,Y -544.700,Z 1349.618,A 0.000,B 0.000,C 90.000,E1 147.248} C_DIS
LIN {X 0.025,Y -546.428,Z 1349.614,A 0.000,B 0.000,C 90.000,E1 146.421} C_DIS
LIN {X -0.161,Y -547.875,Z 1349.609,A 0.000,B 0.000,C 90.000,E1 145.595} C_DIS
LIN {X -0.020,Y -549.077,Z 1349.604,A 0.000,B 0.000,C 90.000,E1 144.736} C_DIS
LIN {X -0.125,Y -550.340,Z 1349.598,A 0.000,B 0.000,C 90.000,E1 143.623} C_DIS
LIN {X 0.049,Y -551.124,Z 1349.593,A 0.000,B 0.000,C 90.000,E1 142.763} C_DIS
LIN {X 0.230,Y -551.735,Z 1349.589,A 0.000,B 0.000,C 90.000,E1 141.904} C_DIS
LIN {X 0.107,Y -552.633,Z 1349.581,A 0.000,B 0.000,C 90.000,E1 140.517} C_DIS
LIN {X -0.009,Y -553.690,Z 1349.571,A 0.000,B 0.000,C 90.000,E1 138.852} C_DIS
LIN {X 0.268,Y -554.658,Z 1349.562,A 0.000,B 0.000,C 90.000,E1 137.148} C_DIS
LIN {X 0.258,Y -555.986,Z 1349.550,A 0.000,B 0.000,C 90.000,E1 134.919} C_DIS
LIN {X -0.080,Y -556.686,Z 1349.546,A 0.000,B 0.000,C 90.000,E1 134.271} C_DIS
LIN {X -0.011,Y -557.597,Z 1349.544,A 0.000,B 0.000,C 90.000,E1 133.866} C_DIS
LIN {X -0.053,Y -557.622,Z 1349.544,A 0.000,B 0.000,C 90.000,E1 133.866} C_DIS
LIN {X 0.016,Y -558.169,Z 1349.543,A 0.000,B 0.000,C 90.000,E1 133.785} C_DIS
LIN {X 0.240,Y -559.940,Z 1349.542,A 0.000,B 0.000,C 90.000,E1 133.623} C_DIS
LIN {X -0.242,Y -561.165,Z 1349.542,A 0.000,B 0.000,C 90.000,E1 133.623} C_DIS
LIN {X -0.017,Y -568.105,Z 1349.541,A 0.000,B 0.000,C 90.000,E1 133.419} C_DIS
LIN {X 0.053,Y -574.363,Z 1349.540,A 0.000,B 0.000,C 90.000,E1 133.218} C_DIS
LIN {X 0.184,Y -577.497,Z 1349.540,A 0.000,B 0.000,C 90.000,E1 133.095} C_DIS
LIN {X -0.080,Y -583.355,Z 1349.538,A 0.000,B 0.000,C 90.000,E1 132.852} C_DIS
LIN {X 0.064,Y -588.977,Z 1349.536,A 0.000,B 0.000,C 90.000,E1 132.486} C_DIS
LIN {X -0.159,Y -593.274,Z 1349.534,A 0.000,B 0.000,C 90.000,E1 132.204} C_DIS
LIN {X -0.025,Y -598.874,Z 1349.532,A 0.000,B 0.000,C 90.000,E1 131.757} C_DIS
LIN {X 0.229,Y -602.910,Z 1349.530,A 0.000,B 0.000,C 90.000,E1 131.391} C_DIS
LIN {X 0.241,Y -609.306,Z 1349.527,A 0.000,B 0.000,C 90.000,E1 130.782} C_DIS
LIN {X -0.272,Y -613.076,Z 1349.525,A 0.000,B 0.000,C 90.000,E1 130.458} C_DIS
LIN {X 0.040,Y -616.796,Z 1349.523,A 0.000,B 0.000,C 90.000,E1 130.048} C_DIS
LIN {X 0.056,Y -623.598,Z 1349.518,A 0.000,B 0.000,C 90.000,E1 129.277} C_DIS
LIN {X -0.296,Y -630.101,Z 1349.514,A 0.000,B 0.000,C 90.000,E1 128.543} C_DIS
LIN {X -0.072,Y -634.225,Z 1349.511,A 0.000,B 0.000,C 90.000,E1 128.016} C_DIS
LIN {X 0.180,Y -640.005,Z 1349.507,A 0.000,B 0.000,C 90.000,E1 127.237} C_DIS
LIN {X -0.002,Y -646.468,Z 1349.502,A 0.000,B 0.000,C 90.000,E1 126.377} C_DIS
LIN {X 0.039,Y -650.994,Z 1349.499,A 0.000,B 0.000,C 90.000,E1 125.758} C_DIS
LIN {X 0.087,Y -657.393,Z 1349.493,A 0.000,B 0.000,C 90.000,E1 124.771} C_DIS
LIN {X 0.011,Y -658.901,Z 1349.492,A 0.000,B 0.000,C 90.000,E1 124.532} C_DIS
LIN {X 0.091,Y -662.336,Z 1349.489,A 0.000,B 0.000,C 90.000,E1 123.913} C_DIS
LIN {X 0.137,Y -664.906,Z 1349.486,A 0.000,B 0.000,C 90.000,E1 123.420} C_DIS
LIN {X -0.166,Y -667.264,Z 1349.483,A 0.000,B 0.000,C 90.000,E1 122.959} C_DIS
LIN {X 0.051,Y -670.260,Z 1349.479,A 0.000,B 0.000,C 90.000,E1 122.212} C_DIS
LIN {X 0.298,Y -672.875,Z 1349.475,A 0.000,B 0.000,C 90.000,E1 121.465} C_DIS
LIN {X -0.184,Y -675.812,Z 1349.470,A 0.000,B 0.000,C 90.000,E1 120.541} C_DIS
LIN {X 0.111,Y -677.540,Z 1349.466,A 0.000,B 0.000,C 90.000,E1 119.795} C_DIS
LIN {X 0.085,Y -678.841,Z 1349.462,A 0.000,B 0.000,C 90.000,E1 119.077} C_DIS
LIN {X 0.072,Y -679.559,Z 1349.458,A 0.000,B 0.000,C 90.000,E1 118.359} C_DIS
LIN {X -0.133,Y -679.807,Z 1349.455,A 0.000,B 0.000,C 90.000,E1 117.897} C_DIS
LIN {X 0.059,Y -679.828,Z 1349.450,A 0.000,B 0.000,C 90.000,E1 116.924} C_DIS
LIN {X -0.254,Y -679.614,Z 1349.446,A 0.000,B 0.000,C 90.000,E1 116.232} C_DIS
LIN {X 0.341,Y -679.153,Z 1349.442,A 0.000,B 0.000,C 90.000,E1 115.463} C_DIS
LIN {X -0.168,Y -678.682,Z 1349.439,A 0.000,B 0.000,C 90.000,E1 115.027} C_DIS
LIN {X 0.222,Y -677.838,Z 1349.436,A 0.000,B 0.000,C 90.000,E1 114.515} C_DIS
LIN {X 0.134,Y -677.237,Z 1349.435,A 0.000,B 0.000,C 90.000,E1 114.283} C_DIS
LIN {X -0.104,Y -675.457,Z 1349.432,A 0.000,B 0.000,C 90.000,E1 113.823} C_DIS
LIN {X -0.013,Y -674.819,Z 1349.432,A 0.000,B 0.000,C 90.000,E1 113.695} C_DIS
LIN {X 0.073,Y -671.234,Z 1349.429,A 0.000,B 0.000,C 90.000,E1 113.206} C_DIS
LIN {X 0.158,Y -670.088,Z 1349.428,A 0.000,B 0.000,C 90.000,E1 113.078} C_DIS
LIN {X 0.297,Y -663.603,Z 1349.426,A 0.000,B 0.000,C 90.000,E1 112.642} C_DIS
LIN {X -0.247,Y -661.775,Z 1349.425,A 0.000,B 0.000,C 90.000,E1 112.589} C_DIS
LIN {X 0.006,Y -657.106,Z 1349.425,A 0.000,B 0.000,C 90.000,E1 112.408} C_DIS
LIN {X 0.222,Y -652.874,Z 1349.424,A 0.000,B 0.000,C 90.000,E1 112.280} C_DIS
LIN {X 0.162,Y -638.076,Z 1349.422,A 0.000,B 0.000,C 90.000,E1 111.972} C_DIS
LIN {X -0.211,Y -637.035,Z 1349.422,A 0.000,B 0.000,C 90.000,E1 111.972} C_DIS
LIN {X -0.026,Y -636.960,Z 1349.422,A 0.000,B 0.000,C 90.000,E1 111.950} C_DIS
LIN {X 0.261,Y -637.910,Z 1349.421,A 0.000,B 0.000,C 90.000,E1 111.770} C_DIS
LIN {X -0.204,Y -645.428,Z 1349.416,A 0.000,B 0.000,C 90.000,E1 110.918} C_DIS
LIN {X -0.265,Y -650.194,Z 1349.413,A 0.000,B 0.000,C 90.000,E1 110.301} C_DIS
LIN {X 0.145,Y -654.704,Z 1349.409,A 0.000,B 0.000,C 90.000,E1 109.523} C_DIS
LIN {X 0.039,Y -659.083,Z 1349.404,A 0.000,B 0.000,C 90.000,E1 108.671} C_DIS
LIN {X -0.079,Y -662.284,Z 1349.400,A 0.000,B 0.000,C 90.000,E1 107.946} C_DIS
LIN {X -0.260,Y -666.154,Z 1349.394,A 0.000,B 0.000,C 90.000,E1 106.985} C_DIS
LIN {X -0.318,Y -668.681,Z 1349.390,A 0.000,B 0.000,C 90.000,E1 106.260} C_DIS
LIN {X 0.286,Y -670.815,Z 1349.386,A 0.000,B 0.000,C 90.000,E1 105.481} C_DIS
LIN {X 0.086,Y -672.535,Z 1349.382,A 0.000,B 0.000,C 90.000,E1 104.773} C_DIS
LIN {X -0.037,Y -673.519,Z 1349.380,A 0.000,B 0.000,C 90.000,E1 104.300} C_DIS
LIN {X -0.152,Y -674.255,Z 1349.377,A 0.000,B 0.000,C 90.000,E1 103.828} C_DIS
LIN {X -0.319,Y -674.938,Z 1349.373,A 0.000,B 0.000,C 90.000,E1 103.119} C_DIS
LIN {X 0.233,Y -675.213,Z 1349.370,A 0.000,B 0.000,C 90.000,E1 102.591} C_DIS
LIN {X 0.070,Y -675.132,Z 1349.366,A 0.000,B 0.000,C 90.000,E1 101.883} C_DIS
LIN {X -0.230,Y -674.676,Z 1349.362,A 0.000,B 0.000,C 90.000,E1 101.186} C_DIS
LIN {X 0.317,Y -674.140,Z 1349.359,A 0.000,B 0.000,C 90.000,E1 100.658} C_DIS
LIN {X 0.074,Y -673.420,Z 1349.357,A 0.000,B 0.000,C 90.000,E1 100.197} C_DIS
LIN {X -0.053,Y -672.406,Z 1349.354,A 0.000,B 0.000,C 90.000,E1 99.726} C_DIS
LIN {X -0.302,Y -671.119,Z 1349.351,A 0.000,B 0.000,C 90.000,E1 99.265} C_DIS
LIN {X 0.108,Y -669.552,Z 1349.349,A 0.000,B 0.000,C 90.000,E1 98.746} C_DIS
LIN {X -0.235,Y -666.721,Z 1349.345,A 0.000,B 0.000,C 90.000,E1 98.049} C_DIS
LIN {X 0.149,Y -664.602,Z 1349.342,A 0.000,B 0.000,C 90.000,E1 97.530} C_DIS
LIN {X -0.151,Y -661.704,Z 1349.339,A 0.000,B 0.000,C 90.000,E1 96.947} C_DIS
LIN {X -0.101,Y -657.212,Z 1349.334,A 0.000,B 0.000,C 90.000,E1 96.087} C_DIS
LIN {X 0.112,Y -653.678,Z 1349.330,A 0.000,B 0.000,C 90.000,E1 95.454} C_DIS
LIN {X 0.295,Y -649.774,Z 1349.327,A 0.000,B 0.000,C 90.000,E1 94.821} C_DIS
LIN {X -0.090,Y -646.499,Z 1349.324,A 0.000,B 0.000,C 90.000,E1 94.359} C_DIS
LIN {X 0.145,Y -642.947,Z 1349.321,A 0.000,B 0.000,C 90.000,E1 93.841} C_DIS
LIN {X -0.327,Y -639.130,Z 1349.319,A 0.000,B 0.000,C 90.000,E1 93.383} C_DIS
LIN {X -0.146,Y -634.639,Z 1349.316,A 0.000,B 0.000,C 90.000,E1 92.865} C_DIS
LIN {X -0.125,Y -624.849,Z 1349.311,A 0.000,B 0.000,C 90.000,E1 91.892} C_DIS
LIN {X -0.055,Y -617.230,Z 1349.306,A 0.000,B 0.000,C 90.000,E1 91.146} C_DIS
LIN {X -0.193,Y -610.455,Z 1349.303,A 0.000,B 0.000,C 90.000,E1 90.573} C_DIS
LIN {X -0.212,Y -608.959,Z 1349.302,A 0.000,B 0.000,C 90.000,E1 90.458} C_DIS
LIN {X 0.186,Y -602.581,Z 1349.300,A 0.000,B 0.000,C 90.000,E1 90.000} C_DIS
LIN {X -0.113,Y -595.519,Z 1349.298,A 0.000,B 0.000,C 90.000,E1 89.656} C_DIS
LIN {X -0.229,Y -581.560,Z 1349.295,A 0.000,B 0.000,C 90.000,E1 89.083} C_DIS
LIN {X -0.025,Y -577.224,Z 1349.294,A 0.000,B 0.000,C 90.000,E1 88.854} C_DIS
LIN {X -0.223,Y -576.085,Z 1349.293,A 0.000,B 0.000,C 90.000,E1 88.797} C_DIS
LIN {X 0.019,Y -573.802,Z 1349.292,A 0.000,B 0.000,C 90.000,E1 88.568} C_DIS
LIN {X -0.205,Y -573.245,Z 1349.292,A 0.000,B 0.000,C 90.000,E1 88.511} C_DIS
LIN {X -0.239,Y -573.224,Z 1349.292,A 0.000,B 0.000,C 90.000,E1 88.511} C_DIS
LIN {X 0.215,Y -572.708,Z 1349.290,A 0.000,B 0.000,C 90.000,E1 88.165} C_DIS
LIN {X 0.062,Y -573.230,Z 1349.285,A 0.000,B 0.000,C 90.000,E1 87.364} C_DIS
LIN {X -0.041,Y -575.026,Z 1349.275,A 0.000,B 0.000,C 90.000,E1 85.469} C_DIS
LIN {X 0.145,Y -577.466,Z 1349.263,A 0.000,B 0.000,C 90.000,E1 83.280} C_DIS
LIN {X 0.254,Y -579.692,Z 1349.252,A 0.000,B 0.000,C 90.000,E1 81.376} C_DIS
LIN {X 0.131,Y -581.332,Z 1349.245,A 0.000,B 0.000,C 90.000,E1 80.038} C_DIS
LIN {X 0.035,Y -582.744,Z 1349.237,A 0.000,B 0.000,C 90.000,E1 78.701} C_DIS
LIN {X 0.075,Y -584.066,Z 1349.230,A 0.000,B 0.000,C 90.000,E1 77.353} C_DIS
LIN {X 0.275,Y -585.197,Z 1349.222,A 0.000,B 0.000,C 90.000,E1 75.992} C_DIS
LIN {X -0.064,Y -586.280,Z 1349.215,A 0.000,B 0.000,C 90.000,E1 74.685} C_DIS
LIN {X 0.176,Y -587.144,Z 1349.208,A 0.000,B 0.000,C 90.000,E1 73.323} C_DIS
LIN {X -0.293,Y -588.111,Z 1349.199,A 0.000,B 0.000,C 90.000,E1 71.764} C_DIS
LIN {X -0.136,Y -589.249,Z 1349.188,A 0.000,B 0.000,C 90.000,E1 69.880} C_DIS
LIN {X 0.259,Y -590.414,Z 1349.178,A 0.000,B 0.000,C 90.000,E1 67.975} C_DIS
LIN {X 0.020,Y -591.948,Z 1349.166,A 0.000,B 0.000,C 90.000,E1 65.869} C_DIS
LIN {X 0.055,Y -593.007,Z 1349.159,A 0.000,B 0.000,C 90.000,E1 64.537} C_DIS
LIN {X 0.013,Y -594.067,Z 1349.150,A 0.000,B 0.000,C 90.000,E1 62.948} C_DIS
LIN {X -0.069,Y -595.551,Z 1349.139,A 0.000,B 0.000,C 90.000,E1 61.101} C_DIS
LIN {X -0.220,Y -596.782,Z 1349.132,A 0.000,B 0.000,C 90.000,E1 59.793} C_DIS
LIN {X -0.052,Y -598.172,Z 1349.125,A 0.000,B 0.000,C 90.000,E1 58.456} C_DIS
LIN {X 0.132,Y -599.448,Z 1349.117,A 0.000,B 0.000,C 90.000,E1 57.120} C_DIS
LIN {X 0.160,Y -600.735,Z 1349.110,A 0.000,B 0.000,C 90.000,E1 55.801} C_DIS
LIN {X 0.211,Y -602.012,Z 1349.103,A 0.000,B 0.000,C 90.000,E1 54.482} C_DIS
LIN {X -0.180,Y -603.760,Z 1349.093,A 0.000,B 0.000,C 90.000,E1 52.683} C_DIS
LIN {X -0.205,Y -604.695,Z 1349.085,A 0.000,B 0.000,C 90.000,E1 51.376} C_DIS
LIN {X 0.036,Y -605.676,Z 1349.077,A 0.000,B 0.000,C 90.000,E1 49.784} C_DIS
LIN {X -0.047,Y -606.264,Z 1349.069,A 0.000,B 0.000,C 90.000,E1 48.485} C_DIS
LIN {X 0.097,Y -606.656,Z 1349.061,A 0.000,B 0.000,C 90.000,E1 46.905} C_DIS
LIN {X 0.067,Y -606.855,Z 1349.051,A 0.000,B 0.000,C 90.000,E1 45.081} C_DIS
LIN {X 0.169,Y -606.682,Z 1349.045,A 0.000,B 0.000,C 90.000,E1 44.028} C_DIS
LIN {X 0.039,Y -606.423,Z 1349.040,A 0.000,B 0.000,C 90.000,E1 43.257} C_DIS
LIN {X 0.184,Y -605.746,Z 1349.032,A 0.000,B 0.000,C 90.000,E1 41.676} C_DIS
LIN {X 0.100,Y -605.053,Z 1349.024,A 0.000,B 0.000,C 90.000,E1 40.378} C_DIS
LIN {X -0.129,Y -604.195,Z 1349.016,A 0.000,B 0.000,C 90.000,E1 38.830} C_DIS
LIN {X 0.174,Y -603.702,Z 1349.011,A 0.000,B 0.000,C 90.000,E1 38.016} C_DIS
LIN {X 0.101,Y -603.071,Z 1349.007,A 0.000,B 0.000,C 90.000,E1 37.237} C_DIS
LIN {X 0.028,Y -602.228,Z 1349.003,A 0.000,B 0.000,C 90.000,E1 36.457} C_DIS
LIN {X 0.048,Y -601.522,Z 1349.000,A 0.000,B 0.000,C 90.000,E1 35.931} C_DIS
LIN {X -0.047,Y -600.262,Z 1348.995,A 0.000,B 0.000,C 90.000,E1 35.152} C_DIS
LIN {X 0.097,Y -599.284,Z 1348.992,A 0.000,B 0.000,C 90.000,E1 34.612} C_DIS
LIN {X -0.122,Y -597.166,Z 1348.987,A 0.000,B 0.000,C 90.000,E1 33.579} C_DIS
LIN {X 0.232,Y -595.321,Z 1348.982,A 0.000,B 0.000,C 90.000,E1 32.752} C_DIS
LIN {X -0.046,Y -592.586,Z 1348.976,A 0.000,B 0.000,C 90.000,E1 31.720} C_DIS
LIN {X -0.169,Y -589.139,Z 1348.970,A 0.000,B 0.000,C 90.000,E1 30.669} C_DIS
LIN {X -0.212,Y -586.393,Z 1348.966,A 0.000,B 0.000,C 90.000,E1 29.873} C_DIS
LIN {X -0.283,Y -583.082,Z 1348.961,A 0.000,B 0.000,C 90.000,E1 29.077} C_DIS
LIN {X 0.049,Y -578.829,Z 1348.956,A 0.000,B 0.000,C 90.000,E1 28.103} C_DIS
LIN {X 0.319,Y -573.942,Z 1348.951,A 0.000,B 0.000,C 90.000,E1 27.129} C_DIS
LIN {X -0.161,Y -569.394,Z 1348.946,A 0.000,B 0.000,C 90.000,E1 26.360} C_DIS
LIN {X -0.083,Y -565.153,Z 1348.943,A 0.000,B 0.000,C 90.000,E1 25.668} C_DIS
LIN {X -0.001,Y -558.776,Z 1348.937,A 0.000,B 0.000,C 90.000,E1 24.695} C_DIS
LIN {X -0.022,Y -553.702,Z 1348.933,A 0.000,B 0.000,C 90.000,E1 24.003} C_DIS
LIN {X -0.303,Y -548.360,Z 1348.930,A 0.000,B 0.000,C 90.000,E1 23.334} C_DIS
LIN {X 0.092,Y -542.586,Z 1348.926,A 0.000,B 0.000,C 90.000,E1 22.589} C_DIS
LIN {X 0.108,Y -535.549,Z 1348.921,A 0.000,B 0.000,C 90.000,E1 21.770} C_DIS
LIN {X 0.119,Y -527.819,Z 1348.916,A 0.000,B 0.000,C 90.000,E1 20.918} C_DIS
LIN {X -0.201,Y -521.199,Z 1348.912,A 0.000,B 0.000,C 90.000,E1 20.248} C_DIS
LIN {X 0.217,Y -510.504,Z 1348.906,A 0.000,B 0.000,C 90.000,E1 19.087} C_DIS
LIN {X 0.006,Y -504.183,Z 1348.902,A 0.000,B 0.000,C 90.000,E1 18.417} C_DIS
LIN {X 0.214,Y -493.192,Z 1348.896,A 0.000,B 0.000,C 90.000,E1 17.275} C_DIS
LIN {X 0.132,Y -484.751,Z 1348.892,A 0.000,B 0.000,C 90.000,E1 16.496} C_DIS
LIN {X -0.139,Y -466.408,Z 1348.882,A 0.000,B 0.000,C 90.000,E1 14.773} C_DIS
LIN {X 0.102,Y -453.406,Z 1348.875,A 0.000,B 0.000,C 90.000,E1 13.480} C_DIS
LIN {X -0.187,Y -436.286,Z 1348.865,A 0.000,B 0.000,C 90.000,E1 11.771} C_DIS
LIN {X -0.052,Y -419.322,Z 1348.855,A 0.000,B 0.000,C 90.000,E1 9.905} C_DIS
LIN {X 0.015,Y -406.608,Z 1348.847,A 0.000,B 0.000,C 90.000,E1 8.454} C_DIS
LIN {X -0.112,Y -398.455,Z 1348.842,A 0.000,B 0.000,C 90.000,E1 7.530} C_DIS
LIN {X -0.037,Y -395.902,Z 1348.840,A 0.000,B 0.000,C 90.000,E1 7.182} C_DIS
LIN {X 0.111,Y -394.319,Z 1348.838,A 0.000,B 0.000,C 90.000,E1 6.891} C_DIS
LIN {X 0.073,Y -394.329,Z 1348.838,A 0.000,B 0.000,C 90.000,E1 6.891} C_DIS
LIN {X -0.092,Y -395.146,Z 1348.838,A 0.000,B 0.000,C 90.000,E1 6.777} C_DIS
LIN {X -0.107,Y -399.775,Z 1348.835,A 0.000,B 0.000,C 90.000,E1 6.372} C_DIS
LIN {X -0.068,Y -413.611,Z 1348.830,A 0.000,B 0.000,C 90.000,E1 5.391} C_DIS
LIN {X -0.112,Y -416.857,Z 1348.829,A 0.000,B 0.000,C 90.000,E1 5.163} C_DIS
LIN {X -0.042,Y -422.957,Z 1348.826,A 0.000,B 0.000,C 90.000,E1 4.645} C_DIS
LIN {X 0.092,Y -428.844,Z 1348.823,A 0.000,B 0.000,C 90.000,E1 4.073} C_DIS
LIN {X 0.188,Y -435.924,Z 1348.819,A 0.000,B 0.000,C 90.000,E1 3.326} C_DIS
LIN {X 0.032,Y -442.787,Z 1348.814,A 0.000,B 0.000,C 90.000,E1 2.579} C_DIS
LIN {X 0.132,Y -449.542,Z 1348.810,A 0.000,B 0.000,C 90.000,E1 1.776} C_DIS
LIN {X -0.042,Y -455.679,Z 1348.806,A 0.000,B 0.000,C 90.000,E1 1.031} C_DIS
LIN {X -0.038,Y -461.680,Z 1348.801,A 0.000,B 0.000,C 90.000,E1 0.229} C_DIS
LIN {X 0.040,Y -467.929,Z 1348.796,A 0.000,B 0.000,C 90.000,E1 359.312} C_DIS
LIN {X 0.164,Y -472.991,Z 1348.792,A 0.000,B 0.000,C 90.000,E1 358.511} C_DIS
LIN {X 0.011,Y -478.473,Z 1348.787,A 0.000,B 0.000,C 90.000,E1 357.593} C_DIS
LIN {X 0.090,Y -481.962,Z 1348.783,A 0.000,B 0.000,C 90.000,E1 356.963} C_DIS
LIN {X -0.114,Y -485.991,Z 1348.779,A 0.000,B 0.000,C 90.000,E1 356.216} C_DIS
LIN {X 0.207,Y -489.617,Z 1348.775,A 0.000,B 0.000,C 90.000,E1 355.412} C_DIS
LIN {X -0.088,Y -492.307,Z 1348.771,A 0.000,B 0.000,C 90.000,E1 354.837} C_DIS
LIN {X 0.193,Y -496.662,Z 1348.765,A 0.000,B 0.000,C 90.000,E1 353.742} C_DIS
LIN {X 0.118,Y -499.486,Z 1348.761,A 0.000,B 0.000,C 90.000,E1 352.996} C_DIS
LIN {X -0.196,Y -502.506,Z 1348.756,A 0.000,B 0.000,C 90.000,E1 352.129} C_DIS
LIN {X 0.037,Y -506.018,Z 1348.750,A 0.000,B 0.000,C 90.000,E1 350.905} C_DIS
LIN {X -0.206,Y -508.301,Z 1348.745,A 0.000,B 0.000,C 90.000,E1 350.038} C_DIS
LIN {X 0.162,Y -510.379,Z 1348.740,A 0.000,B 0.000,C 90.000,E1 349.106} C_DIS
LIN {X 0.022,Y -512.833,Z 1348.733,A 0.000,B 0.000,C 90.000,E1 347.937} C_DIS
LIN {X -0.064,Y -514.445,Z 1348.728,A 0.000,B 0.000,C 90.000,E1 347.061} C_DIS
LIN {X -0.016,Y -515.826,Z 1348.723,A 0.000,B 0.000,C 90.000,E1 346.172} C_DIS
LIN {X 0.053,Y -517.052,Z 1348.718,A 0.000,B 0.000,C 90.000,E1 345.283} C_DIS
LIN {X 0.118,Y -518.206,Z 1348.712,A 0.000,B 0.000,C 90.000,E1 344.102} C_DIS
LIN {X -0.290,Y -518.803,Z 1348.707,A 0.000,B 0.000,C 90.000,E1 343.268} C_DIS
LIN {X -0.043,Y -519.173,Z 1348.702,A 0.000,B 0.000,C 90.000,E1 342.362} C_DIS
LIN {X 0.212,Y -519.245,Z 1348.697,A 0.000,B 0.000,C 90.000,E1 341.456} C_DIS
LIN {X -0.023,Y -519.065,Z 1348.692,A 0.000,B 0.000,C 90.000,E1 340.604} C_DIS
LIN {X 0.087,Y -518.800,Z 1348.689,A 0.000,B 0.000,C 90.000,E1 340.007} C_DIS
LIN {X -0.115,Y -518.308,Z 1348.686,A 0.000,B 0.000,C 90.000,E1 339.444} C_DIS
LIN {X -0.018,Y -517.519,Z 1348.682,A 0.000,B 0.000,C 90.000,E1 338.847} C_DIS
LIN {X 0.121,Y -516.889,Z 1348.681,A 0.000,B 0.000,C 90.000,E1 338.539} C_DIS
LIN {X -0.222,Y -515.989,Z 1348.679,A 0.000,B 0.000,C 90.000,E1 338.284} C_DIS
LIN {X -0.087,Y -514.805,Z 1348.678,A 0.000,B 0.000,C 90.000,E1 337.975} C_DIS
LIN {X 0.218,Y -513.998,Z 1348.677,A 0.000,B 0.000,C 90.000,E1 337.794} C_DIS
LIN {X 0.045,Y -512.944,Z 1348.676,A 0.000,B 0.000,C 90.000,E1 337.667} C_DIS
LIN {X -0.130,Y -510.966,Z 1348.675,A 0.000,B 0.000,C 90.000,E1 337.539} C_DIS
LIN {X 0.114,Y -480.958,Z 1348.667,A 0.000,B 0.000,C 90.000,E1 336.049} C_DIS
LIN {X 0.062,Y -454.427,Z 1348.659,A 0.000,B 0.000,C 90.000,E1 334.588} C_DIS
LIN {X 0.082,Y -429.868,Z 1348.650,A 0.000,B 0.000,C 90.000,E1 333.050} C_DIS
LIN {X 0.034,Y -407.280,Z 1348.641,A 0.000,B 0.000,C 90.000,E1 331.463} C_DIS
LIN {X 0.033,Y -386.641,Z 1348.632,A 0.000,B 0.000,C 90.000,E1 329.822} C_DIS
LIN {X 0.069,Y -368.008,Z 1348.623,A 0.000,B 0.000,C 90.000,E1 328.152} C_DIS
LIN {X 0.040,Y -367.997,Z 1348.623,A 0.000,B 0.000,C 90.000,E1 328.152} C_DIS
LIN {X -0.092,Y -371.771,Z 1348.602,A 0.000,B 0.000,C 90.000,E1 324.276} C_DIS
LIN {X -0.036,Y -377.367,Z 1348.567,A 0.000,B 0.000,C 90.000,E1 318.038} C_DIS
LIN {X -0.038,Y -378.240,Z 1348.563,A 0.000,B 0.000,C 90.000,E1 317.310} C_DIS
LIN {X -0.047,Y -383.950,Z 1348.531,A 0.000,B 0.000,C 90.000,E1 311.515} C_DIS
LIN {X 0.038,Y -384.898,Z 1348.527,A 0.000,B 0.000,C 90.000,E1 310.782} C_DIS
LIN {X 0.212,Y -390.621,Z 1348.495,A 0.000,B 0.000,C 90.000,E1 305.025} C_DIS
LIN {X 0.056,Y -391.115,Z 1348.493,A 0.000,B 0.000,C 90.000,E1 304.692} C_DIS
LIN {X -0.027,Y -391.653,Z 1348.489,A 0.000,B 0.000,C 90.000,E1 303.992} C_DIS
LIN {X -0.131,Y -396.835,Z 1348.459,A 0.000,B 0.000,C 90.000,E1 298.693} C_DIS
LIN {X -0.039,Y -397.287,Z 1348.455,A 0.000,B 0.000,C 90.000,E1 297.975} C_DIS
LIN {X 0.050,Y -401.603,Z 1348.426,A 0.000,B 0.000,C 90.000,E1 292.695} C_DIS
LIN {X 0.171,Y -404.665,Z 1348.395,A 0.000,B 0.000,C 90.000,E1 287.094} C_DIS
LIN {X -0.129,Y -404.735,Z 1348.391,A 0.000,B 0.000,C 90.000,E1 286.441} C_DIS
LIN {X 0.164,Y -406.104,Z 1348.364,A 0.000,B 0.000,C 90.000,E1 281.535} C_DIS
LIN {X 0.184,Y -405.958,Z 1348.360,A 0.000,B 0.000,C 90.000,E1 280.838} C_DIS
LIN {X -0.147,Y -405.683,Z 1348.333,A 0.000,B 0.000,C 90.000,E1 276.024} C_DIS
LIN {X 0.188,Y -405.054,Z 1348.328,A 0.000,B 0.000,C 90.000,E1 274.935} C_DIS
LIN {X -0.110,Y -403.492,Z 1348.304,A 0.000,B 0.000,C 90.000,E1 270.802} C_DIS
LIN {X -0.143,Y -403.284,Z 1348.302,A 0.000,B 0.000,C 90.000,E1 270.458} C_DIS
LIN {X 0.041,Y -398.923,Z 1348.271,A 0.000,B 0.000,C 90.000,E1 264.837} C_DIS
LIN {X -0.090,Y -393.103,Z 1348.242,A 0.000,B 0.000,C 90.000,E1 259.567} C_DIS
LIN {X -0.130,Y -392.828,Z 1348.240,A 0.000,B 0.000,C 90.000,E1 259.218} C_DIS
LIN {X -0.039,Y -386.372,Z 1348.214,A 0.000,B 0.000,C 90.000,E1 254.574} C_DIS
LIN {X -0.076,Y -385.260,Z 1348.208,A 0.000,B 0.000,C 90.000,E1 253.504} C_DIS
LIN {X -0.054,Y -384.754,Z 1348.206,A 0.000,B 0.000,C 90.000,E1 253.142} C_DIS
LIN {X 0.172,Y -377.963,Z 1348.182,A 0.000,B 0.000,C 90.000,E1 248.773} C_DIS
LIN {X -0.094,Y -376.225,Z 1348.174,A 0.000,B 0.000,C 90.000,E1 247.358} C_DIS
LIN {X 0.008,Y -374.930,Z 1348.170,A 0.000,B 0.000,C 90.000,E1 246.613} C_DIS
LIN {X 0.070,Y -368.407,Z 1348.148,A 0.000,B 0.000,C 90.000,E1 242.564} C_DIS
LIN {X 0.048,Y -366.032,Z 1348.137,A 0.000,B 0.000,C 90.000,E1 240.717} C_DIS
LIN {X -0.044,Y -359.186,Z 1348.115,A 0.000,B 0.000,C 90.000,E1 236.628} C_DIS
LIN {X -0.027,Y -355.827,Z 1348.100,A 0.000,B 0.000,C 90.000,E1 233.989} C_DIS
LIN {X -0.221,Y -348.784,Z 1348.075,A 0.000,B 0.000,C 90.000,E1 229.461} C_DIS
LIN {X -0.145,Y -346.177,Z 1348.062,A 0.000,B 0.000,C 90.000,E1 227.148} C_DIS
LIN {X -0.136,Y -345.053,Z 1348.058,A 0.000,B 0.000,C 90.000,E1 226.377} C_DIS
LIN {X 0.047,Y -338.579,Z 1348.030,A 0.000,B 0.000,C 90.000,E1 221.310} C_DIS
LIN {X 0.047,Y -336.831,Z 1348.019,A 0.000,B 0.000,C 90.000,E1 219.358} C_DIS
LIN {X -0.065,Y -332.781,Z 1348.000,A 0.000,B 0.000,C 90.000,E1 216.011} C_DIS
LIN {X -0.083,Y -332.787,Z 1348.000,A 0.000,B 0.000,C 90.000,E1 216.011} C_DIS
LIN {X -0.168,Y -349.470,Z 1347.990,A 0.000,B 0.000,C 90.000,E1 214.119} C_DIS
LIN {X -0.142,Y -368.262,Z 1347.979,A 0.000,B 0.000,C 90.000,E1 212.212} C_DIS
LIN {X 0.050,Y -387.424,Z 1347.969,A 0.000,B 0.000,C 90.000,E1 210.463} C_DIS
LIN {X -0.238,Y -408.528,Z 1347.960,A 0.000,B 0.000,C 90.000,E1 208.821} C_DIS
LIN {X 0.211,Y -431.616,Z 1347.951,A 0.000,B 0.000,C 90.000,E1 207.129} C_DIS
LIN {X 0.119,Y -446.601,Z 1347.946,A 0.000,B 0.000,C 90.000,E1 206.181} C_DIS
LIN {X 0.089,Y -448.375,Z 1347.944,A 0.000,B 0.000,C 90.000,E1 205.976} C_DIS
LIN {X -0.002,Y -450.007,Z 1347.943,A 0.000,B 0.000,C 90.000,E1 205.668} C_DIS
LIN {X 0.065,Y -451.202,Z 1347.941,A 0.000,B 0.000,C 90.000,E1 205.335} C_DIS
LIN {X -0.055,Y -452.119,Z 1347.939,A 0.000,B 0.000,C 90.000,E1 205.027} C_DIS
LIN {X -0.097,Y -453.524,Z 1347.935,A 0.000,B 0.000,C 90.000,E1 204.387} C_DIS
LIN {X 0.101,Y -454.551,Z 1347.932,A 0.000,B 0.000,C 90.000,E1 203.718} C_DIS
LIN {X 0.108,Y -456.826,Z 1347.921,A 0.000,B 0.000,C 90.000,E1 201.791} C_DIS
LIN {X -0.099,Y -458.272,Z 1347.914,A 0.000,B 0.000,C 90.000,E1 200.536} C_DIS
LIN {X -0.238,Y -461.115,Z 1347.900,A 0.000,B 0.000,C 90.000,E1 198.000} C_DIS
LIN {X 0.031,Y -461.773,Z 1347.896,A 0.000,B 0.000,C 90.000,E1 197.330} C_DIS
LIN {X 0.017,Y -463.579,Z 1347.886,A 0.000,B 0.000,C 90.000,E1 195.426} C_DIS
LIN {X -0.161,Y -465.560,Z 1347.873,A 0.000,B 0.000,C 90.000,E1 193.231} C_DIS
LIN {X 0.138,Y -467.381,Z 1347.863,A 0.000,B 0.000,C 90.000,E1 191.299} C_DIS
LIN {X -0.157,Y -468.526,Z 1347.856,A 0.000,B 0.000,C 90.000,E1 190.074} C_DIS
LIN {X -0.050,Y -469.698,Z 1347.849,A 0.000,B 0.000,C 90.000,E1 188.803} C_DIS
LIN {X -0.099,Y -470.863,Z 1347.840,A 0.000,B 0.000,C 90.000,E1 187.239} C_DIS
LIN {X -0.189,Y -471.800,Z 1347.832,A 0.000,B 0.000,C 90.000,E1 185.682} C_DIS
LIN {X -0.024,Y -472.377,Z 1347.821,A 0.000,B 0.000,C 90.000,E1 183.784} C_DIS
LIN {X 0.060,Y -472.519,Z 1347.814,A 0.000,B 0.000,C 90.000,E1 182.522} C_DIS
LIN {X 0.144,Y -472.366,Z 1347.807,A 0.000,B 0.000,C 90.000,E1 181.260} C_DIS
LIN {X -0.038,Y -471.951,Z 1347.802,A 0.000,B 0.000,C 90.000,E1 180.344} C_DIS
LIN {X -0.223,Y -471.317,Z 1347.797,A 0.000,B 0.000,C 90.000,E1 179.427} C_DIS
LIN {X 0.053,Y -470.433,Z 1347.792,A 0.000,B 0.000,C 90.000,E1 178.453} C_DIS
LIN {X 0.102,Y -469.026,Z 1347.785,A 0.000,B 0.000,C 90.000,E1 177.192} C_DIS
LIN {X 0.159,Y -467.100,Z 1347.778,A 0.000,B 0.000,C 90.000,E1 175.927} C_DIS
LIN {X -0.064,Y -465.302,Z 1347.772,A 0.000,B 0.000,C 90.000,E1 175.008} C_DIS
LIN {X -0.057,Y -463.896,Z 1347.769,A 0.000,B 0.000,C 90.000,E1 174.375} C_DIS
LIN {X -0.061,Y -461.887,Z 1347.765,A 0.000,B 0.000,C 90.000,E1 173.742} C_DIS
LIN {X 0.187,Y -460.825,Z 1347.763,A 0.000,B 0.000,C 90.000,E1 173.394} C_DIS
LIN {X -0.207,Y -457.709,Z 1347.759,A 0.000,B 0.000,C 90.000,E1 172.648} C_DIS
LIN {X 0.016,Y -453.137,Z 1347.754,A 0.000,B 0.000,C 90.000,E1 171.659} C_DIS
LIN {X 0.116,Y -447.803,Z 1347.748,A 0.000,B 0.000,C 90.000,E1 170.679} C_DIS
LIN {X -0.219,Y -441.563,Z 1347.743,A 0.000,B 0.000,C 90.000,E1 169.746} C_DIS
LIN {X 0.053,Y -431.384,Z 1347.735,A 0.000,B 0.000,C 90.000,E1 168.229} C_DIS
LIN {X 0.100,Y -414.866,Z 1347.721,A 0.000,B 0.000,C 90.000,E1 165.700} C_DIS
LIN {X -0.063,Y -410.777,Z 1347.717,A 0.000,B 0.000,C 90.000,E1 165.046} C_DIS
LIN {X 0.080,Y -408.127,Z 1347.714,A 0.000,B 0.000,C 90.000,E1 164.519} C_DIS
LIN {X -0.137,Y -406.315,Z 1347.711,A 0.000,B 0.000,C 90.000,E1 164.031} C_DIS
LIN {X -0.080,Y -405.933,Z 1347.710,A 0.000,B 0.000,C 90.000,E1 163.850} C_DIS
LIN {X -0.151,Y -405.471,Z 1347.708,A 0.000,B 0.000,C 90.000,E1 163.504} C_DIS
LIN {X -0.189,Y -405.486,Z 1347.708,A 0.000,B 0.000,C 90.000,E1 163.504} C_DIS
LIN {X -0.001,Y -407.190,Z 1347.706,A 0.000,B 0.000,C 90.000,E1 163.087} C_DIS
LIN {X -0.202,Y -410.477,Z 1347.704,A 0.000,B 0.000,C 90.000,E1 162.725} C_DIS
LIN {X 0.204,Y -415.269,Z 1347.701,A 0.000,B 0.000,C 90.000,E1 162.181} C_DIS
LIN {X 0.057,Y -416.669,Z 1347.700,A 0.000,B 0.000,C 90.000,E1 162.054} C_DIS
LIN {X -0.111,Y -423.639,Z 1347.697,A 0.000,B 0.000,C 90.000,E1 161.456} C_DIS
LIN {X -0.042,Y -444.495,Z 1347.688,A 0.000,B 0.000,C 90.000,E1 159.826} C_DIS
LIN {X 0.126,Y -457.164,Z 1347.683,A 0.000,B 0.000,C 90.000,E1 158.847} C_DIS
LIN {X -0.158,Y -466.405,Z 1347.679,A 0.000,B 0.000,C 90.000,E1 158.156} C_DIS
LIN {X -0.179,Y -475.513,Z 1347.674,A 0.000,B 0.000,C 90.000,E1 157.411} C_DIS
LIN {X 0.155,Y -482.833,Z 1347.671,A 0.000,B 0.000,C 90.000,E1 156.741} C_DIS
LIN {X 0.062,Y -489.984,Z 1347.667,A 0.000,B 0.000,C 90.000,E1 156.102} C_DIS
LIN {X -0.079,Y -494.192,Z 1347.665,A 0.000,B 0.000,C 90.000,E1 155.717} C_DIS
LIN {X -0.015,Y -501.041,Z 1347.661,A 0.000,B 0.000,C 90.000,E1 155.025} C_DIS
LIN {X 0.011,Y -506.387,Z 1347.658,A 0.000,B 0.000,C 90.000,E1 154.460} C_DIS
LIN {X -0.241,Y -512.880,Z 1347.654,A 0.000,B 0.000,C 90.000,E1 153.768} C_DIS
LIN {X 0.234,Y -517.762,Z 1347.651,A 0.000,B 0.000,C 90.000,E1 153.127} C_DIS
LIN {X 0.025,Y -522.191,Z 1347.648,A 0.000,B 0.000,C 90.000,E1 152.564} C_DIS
LIN {X 0.087,Y -526.221,Z 1347.644,A 0.000,B 0.000,C 90.000,E1 151.975} C_DIS
LIN {X 0.181,Y -529.825,Z 1347.641,A 0.000,B 0.000,C 90.000,E1 151.385} C_DIS
LIN {X 0.155,Y -533.483,Z 1347.637,A 0.000,B 0.000,C 90.000,E1 150.667} C_DIS
LIN {X -0.162,Y -535.936,Z 1347.634,A 0.000,B 0.000,C 90.000,E1 150.127} C_DIS
LIN {X 0.004,Y -538.060,Z 1347.631,A 0.000,B 0.000,C 90.000,E1 149.537} C_DIS
LIN {X 0.184,Y -540.810,Z 1347.626,A 0.000,B 0.000,C 90.000,E1 148.663} C_DIS
LIN {X -0.080,Y -542.519,Z 1347.623,A 0.000,B 0.000,C 90.000,E1 148.122} C_DIS
LIN {X 0.150,Y -544.537,Z 1347.618,A 0.000,B 0.000,C 90.000,E1 147.248} C_DIS
LIN {X -0.090,Y -545.744,Z 1347.615,A 0.000,B 0.000,C 90.000,E1 146.707} C_DIS
LIN {X -0.286,Y -547.263,Z 1347.610,A 0.000,B 0.000,C 90.000,E1 145.881} C_DIS
LIN {X -0.154,Y -548.531,Z 1347.606,A 0.000,B 0.000,C 90.000,E1 145.022} C_DIS
LIN {X -0.320,Y -549.555,Z 1347.601,A 0.000,B 0.000,C 90.000,E1 144.196} C_DIS
LIN {X -0.099,Y -550.718,Z 1347.595,A 0.000,B 0.000,C 90.000,E1 143.050} C_DIS
LIN {X 0.138,Y -551.529,Z 1347.589,A 0.000,B 0.000,C 90.000,E1 141.904} C_DIS
LIN {X 0.010,Y -552.400,Z 1347.581,A 0.000,B 0.000,C 90.000,E1 140.517} C_DIS
LIN {X -0.172,Y -553.322,Z 1347.573,A 0.000,B 0.000,C 90.000,E1 139.138} C_DIS
LIN {X -0.271,Y -554.301,Z 1347.564,A 0.000,B 0.000,C 90.000,E1 137.472} C_DIS
LIN {X 0.009,Y -555.375,Z 1347.554,A 0.000,B 0.000,C 90.000,E1 135.769} C_DIS
LIN {X -0.072,Y -555.926,Z 1347.550,A 0.000,B 0.000,C 90.000,E1 135.081} C_DIS
LIN {X -0.258,Y -556.554,Z 1347.549,A 0.000,B 0.000,C 90.000,E1 134.757} C_DIS
LIN {X 0.088,Y -556.930,Z 1347.547,A 0.000,B 0.000,C 90.000,E1 134.352} C_DIS
LIN {X 0.046,Y -556.953,Z 1347.547,A 0.000,B 0.000,C 90.000,E1 134.352} C_DIS
LIN {X 0.184,Y -557.815,Z 1347.546,A 0.000,B 0.000,C 90.000,E1 134.190} C_DIS
LIN {X 0.264,Y -558.968,Z 1347.545,A 0.000,B 0.000,C 90.000,E1 134.109} C_DIS
LIN {X 0.179,Y -560.976,Z 1347.545,A 0.000,B 0.000,C 90.000,E1 134.028} C_DIS
LIN {X -0.079,Y -567.879,Z 1347.544,A 0.000,B 0.000,C 90.000,E1 133.866} C_DIS
LIN {X -0.043,Y -574.022,Z 1347.543,A 0.000,B 0.000,C 90.000,E1 133.662} C_DIS
LIN {X -0.058,Y -580.288,Z 1347.541,A 0.000,B 0.000,C 90.000,E1 133.419} C_DIS
LIN {X -0.157,Y -582.983,Z 1347.541,A 0.000,B 0.000,C 90.000,E1 133.299} C_DIS
LIN {X 0.169,Y -587.195,Z 1347.539,A 0.000,B 0.000,C 90.000,E1 133.014} C_DIS
LIN {X -0.363,Y -591.642,Z 1347.537,A 0.000,B 0.000,C 90.000,E1 132.771} C_DIS
LIN {X -0.036,Y -598.506,Z 1347.535,A 0.000,B 0.000,C 90.000,E1 132.204} C_DIS
LIN {X -0.247,Y -601.294,Z 1347.533,A 0.000,B 0.000,C 90.000,E1 132.000} C_DIS
LIN {X -0.126,Y -606.464,Z 1347.531,A 0.000,B 0.000,C 90.000,E1 131.515} C_DIS
LIN {X -0.254,Y -612.700,Z 1347.527,A 0.000,B 0.000,C 90.000,E1 130.906} C_DIS
LIN {X -0.074,Y -617.557,Z 1347.524,A 0.000,B 0.000,C 90.000,E1 130.378} C_DIS
LIN {X 0.388,Y -624.249,Z 1347.520,A 0.000,B 0.000,C 90.000,E1 129.564} C_DIS
LIN {X 0.044,Y -631.717,Z 1347.515,A 0.000,B 0.000,C 90.000,E1 128.705} C_DIS
LIN {X 0.158,Y -638.545,Z 1347.510,A 0.000,B 0.000,C 90.000,E1 127.810} C_DIS
LIN {X 0.360,Y -645.852,Z 1347.505,A 0.000,B 0.000,C 90.000,E1 126.790} C_DIS
LIN {X -0.196,Y -650.309,Z 1347.501,A 0.000,B 0.000,C 90.000,E1 126.217} C_DIS
LIN {X 0.271,Y -652.891,Z 1347.499,A 0.000,B 0.000,C 90.000,E1 125.804} C_DIS
LIN {X 0.029,Y -656.799,Z 1347.496,A 0.000,B 0.000,C 90.000,E1 125.231} C_DIS
LIN {X -0.006,Y -659.057,Z 1347.494,A 0.000,B 0.000,C 90.000,E1 124.865} C_DIS
LIN {X 0.333,Y -663.121,Z 1347.490,A 0.000,B 0.000,C 90.000,E1 124.119} C_DIS
LIN {X 0.017,Y -665.649,Z 1347.487,A 0.000,B 0.000,C 90.000,E1 123.658} C_DIS
LIN {X -0.338,Y -668.968,Z 1347.483,A 0.000,B 0.000,C 90.000,E1 122.959} C_DIS
LIN {X -0.105,Y -671.799,Z 1347.479,A 0.000,B 0.000,C 90.000,E1 122.212} C_DIS
LIN {X 0.157,Y -674.279,Z 1347.475,A 0.000,B 0.000,C 90.000,E1 121.465} C_DIS
LIN {X -0.309,Y -677.104,Z 1347.470,A 0.000,B 0.000,C 90.000,E1 120.541} C_DIS
LIN {X 0.000,Y -678.736,Z 1347.466,A 0.000,B 0.000,C 90.000,E1 119.795} C_DIS
LIN {X -0.015,Y -679.958,Z 1347.462,A 0.000,B 0.000,C 90.000,E1 119.077} C_DIS
LIN {X -0.216,Y -680.470,Z 1347.459,A 0.000,B 0.000,C 90.000,E1 118.615} C_DIS
LIN {X -0.215,Y -680.898,Z 1347.455,A 0.000,B 0.000,C 90.000,E1 117.897} C_DIS
LIN {X -0.009,Y -680.917,Z 1347.450,A 0.000,B 0.000,C 90.000,E1 116.924} C_DIS
LIN {X -0.313,Y -680.695,Z 1347.446,A 0.000,B 0.000,C 90.000,E1 116.232} C_DIS
LIN {X 0.296,Y -680.260,Z 1347.442,A 0.000,B 0.000,C 90.000,E1 115.463} C_DIS
LIN {X -0.208,Y -679.789,Z 1347.439,A 0.000,B 0.000,C 90.000,E1 115.027} C_DIS
LIN {X 0.189,Y -678.934,Z 1347.436,A 0.000,B 0.000,C 90.000,E1 114.515} C_DIS
LIN {X 0.105,Y -678.390,Z 1347.435,A 0.000,B 0.000,C 90.000,E1 114.283} C_DIS
LIN {X -0.126,Y -676.546,Z 1347.432,A 0.000,B 0.000,C 90.000,E1 113.823} C_DIS
LIN {X -0.033,Y -675.991,Z 1347.432,A 0.000,B 0.000,C 90.000,E1 113.695} C_DIS
LIN {X 0.061,Y -672.417,Z 1347.429,A 0.000,B 0.000,C 90.000,E1 113.206} C_DIS
LIN {X 0.148,Y -671.396,Z 1347.428,A 0.000,B 0.000,C 90.000,E1 113.078} C_DIS
LIN {X 0.231,Y -669.811,Z 1347.428,A 0.000,B 0.000,C 90.000,E1 112.950} C_DIS
LIN {X -0.155,Y -663.362,Z 1347.425,A 0.000,B 0.000,C 90.000,E1 112.589} C_DIS
LIN {X 0.259,Y -661.093,Z 1347.425,A 0.000,B 0.000,C 90.000,E1 112.461} C_DIS
LIN {X 0.090,Y -659.090,Z 1347.425,A 0.000,B 0.000,C 90.000,E1 112.408} C_DIS
LIN {X -0.035,Y -652.504,Z 1347.424,A 0.000,B 0.000,C 90.000,E1 112.259} C_DIS
LIN {X -0.077,Y -637.563,Z 1347.422,A 0.000,B 0.000,C 90.000,E1 111.950} C_DIS
LIN {X -0.137,Y -637.502,Z 1347.422,A 0.000,B 0.000,C 90.000,E1 111.950} C_DIS
LIN {X -0.011,Y -640.624,Z 1347.420,A 0.000,B 0.000,C 90.000,E1 111.535} C_DIS
LIN {X -0.110,Y -645.931,Z 1347.416,A 0.000,B 0.000,C 90.000,E1 110.918} C_DIS
LIN {X -0.168,Y -650.631,Z 1347.413,A 0.000,B 0.000,C 90.000,E1 110.301} C_DIS
LIN {X -0.369,Y -655.148,Z 1347.409,A 0.000,B 0.000,C 90.000,E1 109.577} C_DIS
LIN {X 0.312,Y -658.959,Z 1347.405,A 0.000,B 0.000,C 90.000,E1 108.779} C_DIS
LIN {X 0.035,Y -662.773,Z 1347.400,A 0.000,B 0.000,C 90.000,E1 107.946} C_DIS
LIN {X -0.139,Y -666.573,Z 1347.394,A 0.000,B 0.000,C 90.000,E1 106.985} C_DIS
LIN {X -0.193,Y -669.085,Z 1347.390,A 0.000,B 0.000,C 90.000,E1 106.260} C_DIS
LIN {X -0.230,Y -671.216,Z 1347.386,A 0.000,B 0.000,C 90.000,E1 105.536} C_DIS
LIN {X 0.221,Y -672.969,Z 1347.382,A 0.000,B 0.000,C 90.000,E1 104.773} C_DIS
LIN {X 0.101,Y -673.941,Z 1347.380,A 0.000,B 0.000,C 90.000,E1 104.300} C_DIS
LIN {X -0.012,Y -674.676,Z 1347.377,A 0.000,B 0.000,C 90.000,E1 103.828} C_DIS
LIN {X -0.174,Y -675.383,Z 1347.373,A 0.000,B 0.000,C 90.000,E1 103.119} C_DIS
LIN {X -0.279,Y -675.666,Z 1347.370,A 0.000,B 0.000,C 90.000,E1 102.647} C_DIS
LIN {X 0.223,Y -675.600,Z 1347.366,A 0.000,B 0.000,C 90.000,E1 101.883} C_DIS
LIN {X -0.020,Y -675.363,Z 1347.364,A 0.000,B 0.000,C 90.000,E1 101.422} C_DIS
LIN {X -0.129,Y -674.948,Z 1347.361,A 0.000,B 0.000,C 90.000,E1 100.950} C_DIS
LIN {X -0.368,Y -674.321,Z 1347.358,A 0.000,B 0.000,C 90.000,E1 100.489} C_DIS
LIN {X 0.175,Y -673.493,Z 1347.355,A 0.000,B 0.000,C 90.000,E1 99.962} C_DIS
LIN {X -0.066,Y -672.330,Z 1347.353,A 0.000,B 0.000,C 90.000,E1 99.500} C_DIS
LIN {X -0.134,Y -671.682,Z 1347.351,A 0.000,B 0.000,C 90.000,E1 99.265} C_DIS
LIN {X 0.280,Y -670.119,Z 1347.349,A 0.000,B 0.000,C 90.000,E1 98.746} C_DIS
LIN {X -0.060,Y -667.272,Z 1347.345,A 0.000,B 0.000,C 90.000,E1 98.049} C_DIS
LIN {X -0.331,Y -665.167,Z 1347.342,A 0.000,B 0.000,C 90.000,E1 97.587} C_DIS
LIN {X -0.157,Y -661.029,Z 1347.337,A 0.000,B 0.000,C 90.000,E1 96.720} C_DIS
LIN {X 0.057,Y -657.085,Z 1347.333,A 0.000,B 0.000,C 90.000,E1 95.967} C_DIS
LIN {X -0.347,Y -654.242,Z 1347.330,A 0.000,B 0.000,C 90.000,E1 95.511} C_DIS
LIN {X -0.156,Y -650.344,Z 1347.327,A 0.000,B 0.000,C 90.000,E1 94.878} C_DIS
LIN {X 0.109,Y -647.048,Z 1347.324,A 0.000,B 0.000,C 90.000,E1 94.359} C_DIS
LIN {X -0.295,Y -643.511,Z 1347.322,A 0.000,B 0.000,C 90.000,E1 93.898} C_DIS
LIN {X -0.122,Y -639.708,Z 1347.319,A 0.000,B 0.000,C 90.000,E1 93.383} C_DIS
LIN {X 0.062,Y -635.226,Z 1347.316,A 0.000,B 0.000,C 90.000,E1 92.865} C_DIS
LIN {X 0.155,Y -626.671,Z 1347.311,A 0.000,B 0.000,C 90.000,E1 92.007} C_DIS
LIN {X 0.256,Y -617.956,Z 1347.307,A 0.000,B 0.000,C 90.000,E1 91.146} C_DIS
LIN {X 0.079,Y -609.812,Z 1347.303,A 0.000,B 0.000,C 90.000,E1 90.458} C_DIS
LIN {X -0.189,Y -603.367,Z 1347.300,A 0.000,B 0.000,C 90.000,E1 90.057} C_DIS
LIN {X 0.102,Y -599.785,Z 1347.299,A 0.000,B 0.000,C 90.000,E1 89.828} C_DIS
LIN {X -0.010,Y -595.041,Z 1347.298,A 0.000,B 0.000,C 90.000,E1 89.599} C_DIS
LIN {X 0.148,Y -582.911,Z 1347.295,A 0.000,B 0.000,C 90.000,E1 89.083} C_DIS
LIN {X -0.217,Y -578.364,Z 1347.294,A 0.000,B 0.000,C 90.000,E1 88.912} C_DIS
LIN {X 0.243,Y -577.102,Z 1347.293,A 0.000,B 0.000,C 90.000,E1 88.797} C_DIS
LIN {X -0.072,Y -575.838,Z 1347.293,A 0.000,B 0.000,C 90.000,E1 88.740} C_DIS
LIN {X -0.027,Y -573.935,Z 1347.292,A 0.000,B 0.000,C 90.000,E1 88.568} C_DIS
LIN {X 0.193,Y -573.181,Z 1347.292,A 0.000,B 0.000,C 90.000,E1 88.453} C_DIS
LIN {X -0.097,Y -572.653,Z 1347.290,A 0.000,B 0.000,C 90.000,E1 88.165} C_DIS
LIN {X -0.116,Y -573.045,Z 1347.286,A 0.000,B 0.000,C 90.000,E1 87.478} C_DIS
LIN {X -0.223,Y -574.840,Z 1347.275,A 0.000,B 0.000,C 90.000,E1 85.584} C_DIS
LIN {X -0.038,Y -577.247,Z 1347.263,A 0.000,B 0.000,C 90.000,E1 83.394} C_DIS
LIN {X 0.068,Y -579.491,Z 1347.253,A 0.000,B 0.000,C 90.000,E1 81.489} C_DIS
LIN {X 0.176,Y -581.444,Z 1347.244,A 0.000,B 0.000,C 90.000,E1 79.859} C_DIS
LIN {X 0.087,Y -582.835,Z 1347.236,A 0.000,B 0.000,C 90.000,E1 78.522} C_DIS
LIN {X 0.134,Y -584.114,Z 1347.229,A 0.000,B 0.000,C 90.000,E1 77.173} C_DIS
LIN {X 0.195,Y -585.248,Z 1347.221,A 0.000,B 0.000,C 90.000,E1 75.825} C_DIS
LIN {X 0.172,Y -586.097,Z 1347.215,A 0.000,B 0.000,C 90.000,E1 74.755} C_DIS
LIN {X 0.245,Y -587.166,Z 1347.207,A 0.000,B 0.000,C 90.000,E1 73.142} C_DIS
LIN {X -0.224,Y -588.117,Z 1347.198,A 0.000,B 0.000,C 90.000,E1 71.583} C_DIS
LIN {X 0.263,Y -589.123,Z 1347.189,A 0.000,B 0.000,C 90.000,E1 69.934} C_DIS
LIN {X -0.106,Y -590.274,Z 1347.178,A 0.000,B 0.000,C 90.000,E1 68.103} C_DIS
LIN {X -0.113,Y -591.787,Z 1347.167,A 0.000,B 0.000,C 90.000,E1 65.973} C_DIS
LIN {X 0.113,Y -593.001,Z 1347.158,A 0.000,B 0.000,C 90.000,E1 64.357} C_DIS
LIN {X -0.100,Y -593.908,Z 1347.150,A 0.000,B 0.000,C 90.000,E1 63.050} C_DIS
LIN {X -0.025,Y -595.610,Z 1347.139,A 0.000,B 0.000,C 90.000,E1 60.923} C_DIS
LIN {X -0.093,Y -596.632,Z 1347.133,A 0.000,B 0.000,C 90.000,E1 59.871} C_DIS
LIN {X 0.066,Y -597.975,Z 1347.125,A 0.000,B 0.000,C 90.000,E1 58.535} C_DIS
LIN {X -0.026,Y -599.517,Z 1347.116,A 0.000,B 0.000,C 90.000,E1 56.962} C_DIS
LIN {X -0.328,Y -600.810,Z 1347.109,A 0.000,B 0.000,C 90.000,E1 55.674} C_DIS
LIN {X 0.069,Y -602.095,Z 1347.102,A 0.000,B 0.000,C 90.000,E1 54.322} C_DIS
LIN {X -0.090,Y -603.611,Z 1347.093,A 0.000,B 0.000,C 90.000,E1 52.763} C_DIS
LIN {X -0.120,Y -604.568,Z 1347.086,A 0.000,B 0.000,C 90.000,E1 51.457} C_DIS
LIN {X -0.014,Y -605.239,Z 1347.080,A 0.000,B 0.000,C 90.000,E1 50.400} C_DIS
LIN {X -0.287,Y -605.856,Z 1347.074,A 0.000,B 0.000,C 90.000,E1 49.380} C_DIS
LIN {X -0.167,Y -606.267,Z 1347.068,A 0.000,B 0.000,C 90.000,E1 48.324} C_DIS
LIN {X 0.172,Y -606.562,Z 1347.061,A 0.000,B 0.000,C 90.000,E1 46.986} C_DIS
LIN {X -0.150,Y -606.681,Z 1347.055,A 0.000,B 0.000,C 90.000,E1 45.972} C_DIS
LIN {X -0.049,Y -606.747,Z 1347.050,A 0.000,B 0.000,C 90.000,E1 44.919} C_DIS
LIN {X 0.051,Y -606.548,Z 1347.044,A 0.000,B 0.000,C 90.000,E1 43.866} C_DIS
LIN {X -0.272,Y -606.151,Z 1347.038,A 0.000,B 0.000,C 90.000,E1 42.852} C_DIS
LIN {X 0.059,Y -605.575,Z 1347.031,A 0.000,B 0.000,C 90.000,E1 41.515} C_DIS
LIN {X -0.031,Y -604.901,Z 1347.023,A 0.000,B 0.000,C 90.000,E1 40.216} C_DIS
LIN {X 0.205,Y -604.054,Z 1347.015,A 0.000,B 0.000,C 90.000,E1 38.624} C_DIS
LIN {X 0.032,Y -603.542,Z 1347.010,A 0.000,B 0.000,C 90.000,E1 37.855} C_DIS
LIN {X -0.044,Y -602.867,Z 1347.006,A 0.000,B 0.000,C 90.000,E1 37.076} C_DIS
LIN {X -0.124,Y -601.994,Z 1347.002,A 0.000,B 0.000,C 90.000,E1 36.297} C_DIS
LIN {X 0.038,Y -600.389,Z 1346.996,A 0.000,B 0.000,C 90.000,E1 35.231} C_DIS
LIN {X -0.070,Y -598.917,Z 1346.991,A 0.000,B 0.000,C 90.000,E1 34.452} C_DIS
LIN {X 0.200,Y -596.791,Z 1346.986,A 0.000,B 0.000,C 90.000,E1 33.372} C_DIS
LIN {X -0.274,Y -594.916,Z 1346.981,A 0.000,B 0.000,C 90.000,E1 32.625} C_DIS
LIN {X 0.055,Y -592.871,Z 1346.977,A 0.000,B 0.000,C 90.000,E1 31.799} C_DIS
LIN {X 0.047,Y -590.378,Z 1346.972,A 0.000,B 0.000,C 90.000,E1 31.003} C_DIS
LIN {X 0.196,Y -586.764,Z 1346.966,A 0.000,B 0.000,C 90.000,E1 29.922} C_DIS
LIN {X -0.163,Y -583.508,Z 1346.962,A 0.000,B 0.000,C 90.000,E1 29.155} C_DIS
LIN {X -0.332,Y -579.301,Z 1346.957,A 0.000,B 0.000,C 90.000,E1 28.231} C_DIS
LIN {X 0.021,Y -575.190,Z 1346.952,A 0.000,B 0.000,C 90.000,E1 27.385} C_DIS
LIN {X -0.286,Y -572.285,Z 1346.949,A 0.000,B 0.000,C 90.000,E1 26.873} C_DIS
LIN {X -0.099,Y -569.177,Z 1346.946,A 0.000,B 0.000,C 90.000,E1 26.309} C_DIS
LIN {X 0.316,Y -565.810,Z 1346.943,A 0.000,B 0.000,C 90.000,E1 25.720} C_DIS
LIN {X -0.054,Y -562.201,Z 1346.940,A 0.000,B 0.000,C 90.000,E1 25.207} C_DIS
LIN {X 0.094,Y -558.472,Z 1346.937,A 0.000,B 0.000,C 90.000,E1 24.643} C_DIS
LIN {X 0.075,Y -553.384,Z 1346.933,A 0.000,B 0.000,C 90.000,E1 23.951} C_DIS
LIN {X 0.008,Y -548.030,Z 1346.929,A 0.000,B 0.000,C 90.000,E1 23.259} C_DIS
LIN {X -0.107,Y -542.203,Z 1346.925,A 0.000,B 0.000,C 90.000,E1 22.567} C_DIS
LIN {X 0.059,Y -536.156,Z 1346.921,A 0.000,B 0.000,C 90.000,E1 21.844} C_DIS
LIN {X 0.025,Y -531.044,Z 1346.918,A 0.000,B 0.000,C 90.000,E1 21.280} C_DIS
LIN {X 0.245,Y -523.361,Z 1346.914,A 0.000,B 0.000,C 90.000,E1 20.429} C_DIS
LIN {X 0.164,Y -512.711,Z 1346.907,A 0.000,B 0.000,C 90.000,E1 19.322} C_DIS
LIN {X 0.157,Y -503.769,Z 1346.902,A 0.000,B 0.000,C 90.000,E1 18.362} C_DIS
LIN {X -0.215,Y -492.616,Z 1346.896,A 0.000,B 0.000,C 90.000,E1 17.275} C_DIS
LIN {X 0.028,Y -483.937,Z 1346.891,A 0.000,B 0.000,C 90.000,E1 16.441} C_DIS
LIN {X -0.283,Y -469.848,Z 1346.884,A 0.000,B 0.000,C 90.000,E1 15.134} C_DIS
LIN {X 0.121,Y -461.125,Z 1346.879,A 0.000,B 0.000,C 90.000,E1 14.245} C_DIS
LIN {X 0.093,Y -442.655,Z 1346.869,A 0.000,B 0.000,C 90.000,E1 12.411} C_DIS
LIN {X 0.085,Y -421.399,Z 1346.856,A 0.000,B 0.000,C 90.000,E1 10.141} C_DIS
LIN {X -0.057,Y -407.321,Z 1346.848,A 0.000,B 0.000,C 90.000,E1 8.568} C_DIS
LIN {X 0.000,Y -398.844,Z 1346.842,A 0.000,B 0.000,C 90.000,E1 7.587} C_DIS
LIN {X 0.081,Y -396.197,Z 1346.840,A 0.000,B 0.000,C 90.000,E1 7.239} C_DIS
LIN {X -0.147,Y -394.534,Z 1346.839,A 0.000,B 0.000,C 90.000,E1 6.947} C_DIS
LIN {X 0.207,Y -394.542,Z 1346.839,A 0.000,B 0.000,C 90.000,E1 6.891} C_DIS
LIN {X 0.155,Y -395.297,Z 1346.838,A 0.000,B 0.000,C 90.000,E1 6.777} C_DIS
LIN {X 0.066,Y -399.420,Z 1346.836,A 0.000,B 0.000,C 90.000,E1 6.429} C_DIS
LIN {X 0.101,Y -406.643,Z 1346.833,A 0.000,B 0.000,C 90.000,E1 5.910} C_DIS
LIN {X 0.177,Y -413.128,Z 1346.830,A 0.000,B 0.000,C 90.000,E1 5.454} C_DIS
LIN {X 0.186,Y -416.407,Z 1346.829,A 0.000,B 0.000,C 90.000,E1 5.220} C_DIS
LIN {X -0.011,Y -422.434,Z 1346.827,A 0.000,B 0.000,C 90.000,E1 4.759} C_DIS
LIN {X 0.035,Y -429.801,Z 1346.823,A 0.000,B 0.000,C 90.000,E1 4.073} C_DIS
LIN {X 0.106,Y -436.898,Z 1346.819,A 0.000,B 0.000,C 90.000,E1 3.326} C_DIS
LIN {X -0.210,Y -442.499,Z 1346.815,A 0.000,B 0.000,C 90.000,E1 2.751} C_DIS
LIN {X -0.045,Y -449.262,Z 1346.811,A 0.000,B 0.000,C 90.000,E1 1.949} C_DIS
LIN {X 0.005,Y -455.749,Z 1346.806,A 0.000,B 0.000,C 90.000,E1 1.146} C_DIS
LIN {X 0.113,Y -463.023,Z 1346.801,A 0.000,B 0.000,C 90.000,E1 0.172} C_DIS
LIN {X 0.046,Y -468.991,Z 1346.796,A 0.000,B 0.000,C 90.000,E1 359.312} C_DIS
LIN {X 0.180,Y -474.045,Z 1346.792,A 0.000,B 0.000,C 90.000,E1 358.511} C_DIS
LIN {X 0.040,Y -479.535,Z 1346.787,A 0.000,B 0.000,C 90.000,E1 357.593} C_DIS
LIN {X 0.127,Y -483.014,Z 1346.783,A 0.000,B 0.000,C 90.000,E1 356.963} C_DIS
LIN {X -0.220,Y -486.294,Z 1346.780,A 0.000,B 0.000,C 90.000,E1 356.388} C_DIS
LIN {X 0.106,Y -489.973,Z 1346.776,A 0.000,B 0.000,C 90.000,E1 355.584} C_DIS
LIN {X -0.022,Y -493.333,Z 1346.771,A 0.000,B 0.000,C 90.000,E1 354.837} C_DIS
LIN {X -0.221,Y -497.729,Z 1346.766,A 0.000,B 0.000,C 90.000,E1 353.799} C_DIS
LIN {X 0.209,Y -500.539,Z 1346.761,A 0.000,B 0.000,C 90.000,E1 352.996} C_DIS
LIN {X -0.093,Y -503.574,Z 1346.756,A 0.000,B 0.000,C 90.000,E1 352.129} C_DIS
LIN {X 0.157,Y -507.135,Z 1346.750,A 0.000,B 0.000,C 90.000,E1 350.905} C_DIS
LIN {X -0.117,Y -510.104,Z 1346.743,A 0.000,B 0.000,C 90.000,E1 349.746} C_DIS
LIN {X -0.228,Y -512.148,Z 1346.738,A 0.000,B 0.000,C 90.000,E1 348.870} C_DIS
LIN {X 0.159,Y -514.514,Z 1346.732,A 0.000,B 0.000,C 90.000,E1 347.645} C_DIS
LIN {X 0.209,Y -516.057,Z 1346.727,A 0.000,B 0.000,C 90.000,E1 346.756} C_DIS
LIN {X 0.140,Y -517.768,Z 1346.720,A 0.000,B 0.000,C 90.000,E1 345.589} C_DIS
LIN {X 0.241,Y -518.492,Z 1346.717,A 0.000,B 0.000,C 90.000,E1 344.991} C_DIS
LIN {X -0.176,Y -519.612,Z 1346.710,A 0.000,B 0.000,C 90.000,E1 343.866} C_DIS
LIN {X 0.062,Y -520.230,Z 1346.704,A 0.000,B 0.000,C 90.000,E1 342.670} C_DIS
LIN {X -0.024,Y -520.427,Z 1346.697,A 0.000,B 0.000,C 90.000,E1 341.511} C_DIS
LIN {X 0.247,Y -520.216,Z 1346.693,A 0.000,B 0.000,C 90.000,E1 340.604} C_DIS
LIN {X -0.123,Y -519.971,Z 1346.689,A 0.000,B 0.000,C 90.000,E1 340.061} C_DIS
LIN {X 0.172,Y -519.512,Z 1346.686,A 0.000,B 0.000,C 90.000,E1 339.444} C_DIS
LIN {X -0.062,Y -518.530,Z 1346.681,A 0.000,B 0.000,C 90.000,E1 338.592} C_DIS
LIN {X 0.224,Y -517.399,Z 1346.678,A 0.000,B 0.000,C 90.000,E1 337.975} C_DIS
LIN {X -0.116,Y -516.586,Z 1346.676,A 0.000,B 0.000,C 90.000,E1 337.720} C_DIS
LIN {X -0.148,Y -515.039,Z 1346.674,A 0.000,B 0.000,C 90.000,E1 337.283} C_DIS
LIN {X 0.156,Y -514.329,Z 1346.673,A 0.000,B 0.000,C 90.000,E1 337.102} C_DIS
LIN {X -0.017,Y -513.441,Z 1346.672,A 0.000,B 0.000,C 90.000,E1 336.975} C_DIS
LIN {X 0.282,Y -512.211,Z 1346.671,A 0.000,B 0.000,C 90.000,E1 336.794} C_DIS
LIN {X 0.107,Y -509.641,Z 1346.671,A 0.000,B 0.000,C 90.000,E1 336.666} C_DIS
LIN {X -0.092,Y -479.924,Z 1346.662,A 0.000,B 0.000,C 90.000,E1 335.177} C_DIS
LIN {X 0.040,Y -453.591,Z 1346.654,A 0.000,B 0.000,C 90.000,E1 333.640} C_DIS
LIN {X 0.218,Y -429.241,Z 1346.645,A 0.000,B 0.000,C 90.000,E1 332.025} C_DIS
LIN {X -0.054,Y -406.870,Z 1346.636,A 0.000,B 0.000,C 90.000,E1 330.411} C_DIS
LIN {X -0.237,Y -386.455,Z 1346.626,A 0.000,B 0.000,C 90.000,E1 328.742} C_DIS
LIN {X 0.195,Y -368.903,Z 1346.617,A 0.000,B 0.000,C 90.000,E1 327.041} C_DIS
LIN {X 0.165,Y -368.879,Z 1346.617,A 0.000,B 0.000,C 90.000,E1 327.041} C_DIS
LIN {X -0.048,Y -371.641,Z 1346.602,A 0.000,B 0.000,C 90.000,E1 324.402} C_DIS
LIN {X 0.010,Y -376.746,Z 1346.570,A 0.000,B 0.000,C 90.000,E1 318.528} C_DIS
LIN {X -0.235,Y -378.141,Z 1346.564,A 0.000,B 0.000,C 90.000,E1 317.472} C_DIS
LIN {X 0.039,Y -384.263,Z 1346.529,A 0.000,B 0.000,C 90.000,E1 311.272} C_DIS
LIN {X 0.081,Y -384.768,Z 1346.527,A 0.000,B 0.000,C 90.000,E1 310.906} C_DIS
LIN {X 0.071,Y -390.934,Z 1346.494,A 0.000,B 0.000,C 90.000,E1 304.818} C_DIS
LIN {X -0.083,Y -391.358,Z 1346.492,A 0.000,B 0.000,C 90.000,E1 304.485} C_DIS
LIN {X 0.088,Y -397.067,Z 1346.458,A 0.000,B 0.000,C 90.000,E1 298.437} C_DIS
LIN {X 0.044,Y -401.471,Z 1346.427,A 0.000,B 0.000,C 90.000,E1 292.823} C_DIS
LIN {X 0.125,Y -401.680,Z 1346.425,A 0.000,B 0.000,C 90.000,E1 292.461} C_DIS
